LIN {X 0,Y 552.727,Z 232.102,A -85,B 0,C 180,E1 25516.002,E2 25516.002} C_VEL
LIN {X 0,Y 555.255,Z 236.797,A -85,B 0,C 180,E1 25515.534,E2 25515.534} C_VEL
LIN {X 0,Y 562.357,Z 248.705,A -85,B 0,C 180,E1 25514.312,E2 25514.312} C_VEL
LIN {X 0,Y 564.451,Z 252.523,A -85,B 0,C 180,E1 25513.903,E2 25513.903} C_VEL
LIN {X 0,Y 562.986,Z 312.412,A -85,B 0,C 180,E1 25510.976,E2 25510.976} C_VEL
LIN {X 0,Y 564.162,Z 323.504,A -85,B 0,C 180,E1 25510.685,E2 25510.685} C_VEL
LIN {X 0,Y 562.341,Z 534.473,A -85,B 0,C 180,E1 25507.441,E2 25507.441} C_VEL
LIN {X 0,Y 561.246,Z 663.193,A -85,B 0,C 180,E1 25505.485,E2 25505.485} C_VEL
LIN {X 0,Y 560.691,Z 686.814,A -85,B 0,C 180,E1 25504.937,E2 25504.937} C_VEL
LIN {X 0,Y 560.116,Z 709.07,A -85,B 0,C 180,E1 25504.231,E2 25504.231} C_VEL
LIN {X 0,Y 559.344,Z 730.722,A -85,B 0,C 180,E1 25503.343,E2 25503.343} C_VEL
LIN {X 0,Y 558.543,Z 751.818,A -85,B 0,C 180,E1 25502.298,E2 25502.298} C_VEL
LIN {X 0,Y 557.68,Z 772.074,A -85,B 0,C 180,E1 25501.086,E2 25501.086} C_VEL
LIN {X 0,Y 556.797,Z 791.954,A -85,B 0,C 180,E1 25499.709,E2 25499.709} C_VEL
LIN {X 0,Y 555.937,Z 810.881,A -85,B 0,C 180,E1 25498.176,E2 25498.176} C_VEL
LIN {X 0,Y 555.05,Z 830.364,A -85,B 0,C 180,E1 25496.36,E2 25496.36} C_VEL
LIN {X 0,Y 554.323,Z 847.686,A -85,B 0,C 180,E1 25494.509,E2 25494.509} C_VEL
LIN {X 0,Y 553.67,Z 863.855,A -85,B 0,C 180,E1 25492.509,E2 25492.509} C_VEL
LIN {X 0,Y 553.104,Z 879.347,A -85,B 0,C 180,E1 25490.308,E2 25490.308} C_VEL
LIN {X 0,Y 552.685,Z 892.647,A -85,B 0,C 180,E1 25488.128,E2 25488.128} C_VEL
LIN {X 0,Y 552.387,Z 903.847,A -85,B 0,C 180,E1 25485.968,E2 25485.968} C_VEL
LIN {X 0,Y 552.185,Z 913.887,A -85,B 0,C 180,E1 25483.72,E2 25483.72} C_VEL
LIN {X 0,Y 552.045,Z 922.058,A -85,B 0,C 180,E1 25481.491,E2 25481.491} C_VEL
LIN {X 0,Y 551.974,Z 929.049,A -85,B 0,C 180,E1 25479.169,E2 25479.169} C_VEL
LIN {X 0,Y 551.924,Z 934.179,A -85,B 0,C 180,E1 25476.905,E2 25476.905} C_VEL
LIN {X 0,Y 551.901,Z 938.05,A -85,B 0,C 180,E1 25474.571,E2 25474.571} C_VEL
LIN {X 0,Y 551.905,Z 940.19,A -85,B 0,C 180,E1 25472.283,E2 25472.283} C_VEL
LIN {X 0,Y 551.91,Z 940.984,A -85,B 0,C 180,E1 25469.895,E2 25469.895} C_VEL
LIN {X 0,Y 551.905,Z 940.122,A -85,B 0,C 180,E1 25467.611,E2 25467.611} C_VEL
LIN {X 0,Y 551.901,Z 937.911,A -85,B 0,C 180,E1 25465.323,E2 25465.323} C_VEL
LIN {X 0,Y 551.926,Z 934.045,A -85,B 0,C 180,E1 25463.027,E2 25463.027} C_VEL
LIN {X 0,Y 551.977,Z 928.772,A -85,B 0,C 180,E1 25460.722,E2 25460.722} C_VEL
LIN {X 0,Y 552.051,Z 921.694,A -85,B 0,C 180,E1 25458.401,E2 25458.401} C_VEL
LIN {X 0,Y 552.196,Z 912.955,A -85,B 0,C 180,E1 25456.056,E2 25456.056} C_VEL
LIN {X 0,Y 552.397,Z 903.317,A -85,B 0,C 180,E1 25453.922,E2 25453.922} C_VEL
LIN {X 0,Y 552.712,Z 891.365,A -85,B 0,C 180,E1 25451.652,E2 25451.652} C_VEL
LIN {X 0,Y 553.126,Z 878.623,A -85,B 0,C 180,E1 25449.581,E2 25449.581} C_VEL
LIN {X 0,Y 553.701,Z 862.989,A -85,B 0,C 180,E1 25447.378,E2 25447.378} C_VEL
LIN {X 0,Y 554.368,Z 846.587,A -85,B 0,C 180,E1 25445.369,E2 25445.369} C_VEL
LIN {X 0,Y 555.074,Z 829.786,A -85,B 0,C 180,E1 25443.581,E2 25443.581} C_VEL
LIN {X 0,Y 555.964,Z 810.256,A -85,B 0,C 180,E1 25441.771,E2 25441.771} C_VEL
LIN {X 0,Y 556.836,Z 791.177,A -85,B 0,C 180,E1 25440.231,E2 25440.231} C_VEL
LIN {X 0,Y 557.719,Z 771.141,A -85,B 0,C 180,E1 25438.854,E2 25438.854} C_VEL
LIN {X 0,Y 558.61,Z 749.547,A -85,B 0,C 180,E1 25437.582,E2 25437.582} C_VEL
LIN {X 0,Y 559.414,Z 729.067,A -85,B 0,C 180,E1 25436.583,E2 25436.583} C_VEL
LIN {X 0,Y 560.162,Z 706.296,A -85,B 0,C 180,E1 25435.673,E2 25435.673} C_VEL
LIN {X 0,Y 560.75,Z 685.166,A -85,B 0,C 180,E1 25435.018,E2 25435.018} C_VEL
LIN {X 0,Y 561.258,Z 661.984,A -85,B 0,C 180,E1 25434.493,E2 25434.493} C_VEL
LIN {X 0,Y 563.081,Z 445.342,A -85,B 0,C 180,E1 25431.201,E2 25431.201} C_VEL
LIN {X 0,Y 564.019,Z 320.67,A -85,B 0,C 180,E1 25429.256,E2 25429.256} C_VEL
LIN {X 0,Y 562.94,Z 311.331,A -85,B 0,C 180,E1 25428.982,E2 25428.982} C_VEL
LIN {X 0,Y 564.451,Z 252.523,A -85,B 0,C 180,E1 25426.097,E2 25426.097} C_VEL
LIN {X 0,Y 557.462,Z 240.492,A -85,B 0,C 180,E1 25424.82,E2 25424.82} C_VEL
LIN {X 0,Y 553.879,Z 234.143,A -85,B 0,C 180,E1 25424.171,E2 25424.171} C_VEL
LIN {X 0,Y 552.316,Z 230.647,A -85,B 0,C 180,E1 25423.789,E2 25423.789} C_VEL
LIN {X 0,Y 552.267,Z 230.221,A -85,B 0,C 180,E1 25423.296,E2 25423.296} C_VEL
LIN {X 0,Y 552.269,Z 230.249,A -85,B 0,C 180,E1 25419.994,E2 25419.994} C_VEL
LIN {X 0,Y 552.295,Z 230.247,A -85,B 0,C 180,E1 25416.945,E2 25416.945} C_VEL
LIN {X 0,Y 552.268,Z 230.252,A -85,B 0,C 180,E1 25413.642,E2 25413.642} C_VEL
LIN {X 0,Y 552.343,Z 230.249,A -85,B 0,C 180,E1 25410.455,E2 25410.455} C_VEL
LIN {X 0,Y 552.273,Z 230.251,A -85,B 0,C 180,E1 25407.26,E2 25407.26} C_VEL
LIN {X 0,Y 552.324,Z 230.248,A -85,B 0,C 180,E1 25404.036,E2 25404.036} C_VEL
LIN {X 0,Y 552.287,Z 230.248,A -85,B 0,C 180,E1 25400.895,E2 25400.895} C_VEL
LIN {X 0,Y 552.288,Z 230.247,A -85,B 0,C 180,E1 25397.43,E2 25397.43} C_VEL
LIN {X 0,Y 552.339,Z 230.243,A -85,B 0,C 180,E1 25394.252,E2 25394.252} C_VEL
LIN {X 0,Y 552.286,Z 230.246,A -85,B 0,C 180,E1 25390.958,E2 25390.958} C_VEL
LIN {X 0,Y 552.34,Z 230.243,A -85,B 0,C 180,E1 25387.699,E2 25387.699} C_VEL
LIN {X 0,Y 552.304,Z 230.245,A -85,B 0,C 180,E1 25384.465,E2 25384.465} C_VEL
LIN {X 0,Y 552.3,Z 230.238,A -85,B 0,C 180,E1 25381.038,E2 25381.038} C_VEL
LIN {X 0,Y 552.342,Z 230.244,A -85,B 0,C 180,E1 25377.774,E2 25377.774} C_VEL
LIN {X 0,Y 552.301,Z 230.245,A -85,B 0,C 180,E1 25374.495,E2 25374.495} C_VEL
LIN {X 0,Y 552.332,Z 230.236,A -85,B 0,C 180,E1 25371.149,E2 25371.149} C_VEL
LIN {X 0,Y 552.338,Z 230.247,A -85,B 0,C 180,E1 25367.773,E2 25367.773} C_VEL
LIN {X 0,Y 552.307,Z 230.243,A -85,B 0,C 180,E1 25364.459,E2 25364.459} C_VEL
LIN {X 0,Y 552.34,Z 230.235,A -85,B 0,C 180,E1 25361.203,E2 25361.203} C_VEL
LIN {X 0,Y 552.324,Z 230.248,A -85,B 0,C 180,E1 25357.881,E2 25357.881} C_VEL
LIN {X 0,Y 552.322,Z 230.24,A -85,B 0,C 180,E1 25354.479,E2 25354.479} C_VEL
LIN {X 0,Y 552.34,Z 230.241,A -85,B 0,C 180,E1 25352.776,E2 25352.776} C_VEL
LIN {X 0,Y 551.359,Z 230.367,A -85,B 0,C 180,E1 25351.977,E2 25351.977} C_VEL
LIN {X 0,Y 544.843,Z 231.184,A -85,B 0,C 180,E1 25349.675,E2 25349.675} C_VEL
LIN {X 0,Y 544.396,Z 231.235,A -85,B 0,C 180,E1 25349.149,E2 25349.149} C_VEL
LIN {X 0,Y 544.387,Z 231.233,A -85,B 0,C 180,E1 25345.742,E2 25345.742} C_VEL
LIN {X 0,Y 544.395,Z 231.23,A -85,B 0,C 180,E1 25342.295,E2 25342.295} C_VEL
LIN {X 0,Y 544.391,Z 231.235,A -85,B 0,C 180,E1 25338.89,E2 25338.89} C_VEL
LIN {X 0,Y 544.389,Z 231.229,A -85,B 0,C 180,E1 25335.593,E2 25335.593} C_VEL
LIN {X 0,Y 544.399,Z 231.227,A -85,B 0,C 180,E1 25332.238,E2 25332.238} C_VEL
LIN {X 0,Y 544.387,Z 231.234,A -85,B 0,C 180,E1 25328.779,E2 25328.779} C_VEL
LIN {X 0,Y 544.393,Z 231.234,A -85,B 0,C 180,E1 25325.478,E2 25325.478} C_VEL
LIN {X 0,Y 544.39,Z 231.232,A -85,B 0,C 180,E1 25322.147,E2 25322.147} C_VEL
LIN {X 0,Y 544.385,Z 231.238,A -85,B 0,C 180,E1 25318.645,E2 25318.645} C_VEL
LIN {X 0,Y 544.397,Z 231.232,A -85,B 0,C 180,E1 25315.338,E2 25315.338} C_VEL
LIN {X 0,Y 544.375,Z 231.209,A -85,B 0,C 180,E1 25312.006,E2 25312.006} C_VEL
LIN {X 0,Y 544.383,Z 231.233,A -85,B 0,C 180,E1 25308.528,E2 25308.528} C_VEL
LIN {X 0,Y 544.401,Z 231.228,A -85,B 0,C 180,E1 25305.118,E2 25305.118} C_VEL
LIN {X 0,Y 544.37,Z 231.209,A -85,B 0,C 180,E1 25301.774,E2 25301.774} C_VEL
LIN {X 0,Y 544.447,Z 231.538,A -85,B 0,C 180,E1 25301.255,E2 25301.255} C_VEL
LIN {X 0,Y 545.979,Z 235.096,A -85,B 0,C 180,E1 25300.825,E2 25300.825} C_VEL
LIN {X 0,Y 553.743,Z 252.148,A -85,B 0,C 180,E1 25299.008,E2 25299.008} C_VEL
LIN {X 0,Y 551.806,Z 305.653,A -85,B 0,C 180,E1 25295.668,E2 25295.668} C_VEL
LIN {X 0,Y 550.042,Z 360.38,A -85,B 0,C 180,E1 25292.345,E2 25292.345} C_VEL
LIN {X 0,Y 548.57,Z 416.762,A -85,B 0,C 180,E1 25289.006,E2 25289.006} C_VEL
LIN {X 0,Y 549.487,Z 426.879,A -85,B 0,C 180,E1 25288.789,E2 25288.789} C_VEL
LIN {X 0,Y 547.988,Z 628.997,A -85,B 0,C 180,E1 25285.906,E2 25285.906} C_VEL
LIN {X 0,Y 547.682,Z 647.765,A -85,B 0,C 180,E1 25285.445,E2 25285.445} C_VEL
LIN {X 0,Y 547.303,Z 665.668,A -85,B 0,C 180,E1 25284.813,E2 25284.813} C_VEL
LIN {X 0,Y 546.844,Z 682.777,A -85,B 0,C 180,E1 25284.019,E2 25284.019} C_VEL
LIN {X 0,Y 546.339,Z 699.932,A -85,B 0,C 180,E1 25283.011,E2 25283.011} C_VEL
LIN {X 0,Y 545.837,Z 716.086,A -85,B 0,C 180,E1 25281.84,E2 25281.84} C_VEL
LIN {X 0,Y 545.354,Z 731.27,A -85,B 0,C 180,E1 25280.504,E2 25280.504} C_VEL
LIN {X 0,Y 544.923,Z 745.434,A -85,B 0,C 180,E1 25279,E2 25279} C_VEL
LIN {X 0,Y 544.573,Z 758.1,A -85,B 0,C 180,E1 25277.381,E2 25277.381} C_VEL
LIN {X 0,Y 544.3,Z 769.323,A -85,B 0,C 180,E1 25275.643,E2 25275.643} C_VEL
LIN {X 0,Y 544.122,Z 778.555,A -85,B 0,C 180,E1 25273.892,E2 25273.892} C_VEL
LIN {X 0,Y 544,Z 786.466,A -85,B 0,C 180,E1 25272.016,E2 25272.016} C_VEL
LIN {X 0,Y 543.946,Z 792.587,A -85,B 0,C 180,E1 25270.121,E2 25270.121} C_VEL
LIN {X 0,Y 543.915,Z 797.083,A -85,B 0,C 180,E1 25268.172,E2 25268.172} C_VEL
LIN {X 0,Y 543.916,Z 799.805,A -85,B 0,C 180,E1 25266.262,E2 25266.262} C_VEL
LIN {X 0,Y 543.913,Z 800.941,A -85,B 0,C 180,E1 25264.255,E2 25264.255} C_VEL
LIN {X 0,Y 543.911,Z 800.358,A -85,B 0,C 180,E1 25262.286,E2 25262.286} C_VEL
LIN {X 0,Y 543.914,Z 798.153,A -85,B 0,C 180,E1 25260.365,E2 25260.365} C_VEL
LIN {X 0,Y 543.933,Z 794.203,A -85,B 0,C 180,E1 25258.408,E2 25258.408} C_VEL
LIN {X 0,Y 543.974,Z 788.738,A -85,B 0,C 180,E1 25256.537,E2 25256.537} C_VEL
LIN {X 0,Y 544.075,Z 781.346,A -85,B 0,C 180,E1 25254.63,E2 25254.63} C_VEL
LIN {X 0,Y 544.237,Z 772.416,A -85,B 0,C 180,E1 25252.814,E2 25252.814} C_VEL
LIN {X 0,Y 544.471,Z 762.018,A -85,B 0,C 180,E1 25251.096,E2 25251.096} C_VEL
LIN {X 0,Y 544.794,Z 749.92,A -85,B 0,C 180,E1 25249.446,E2 25249.446} C_VEL
LIN {X 0,Y 545.205,Z 736.375,A -85,B 0,C 180,E1 25247.912,E2 25247.912} C_VEL
LIN {X 0,Y 545.673,Z 721.557,A -85,B 0,C 180,E1 25246.518,E2 25246.518} C_VEL
LIN {X 0,Y 546.19,Z 705.24,A -85,B 0,C 180,E1 25245.256,E2 25245.256} C_VEL
LIN {X 0,Y 546.683,Z 688.447,A -85,B 0,C 180,E1 25244.199,E2 25244.199} C_VEL
LIN {X 0,Y 547.148,Z 671.418,A -85,B 0,C 180,E1 25243.341,E2 25243.341} C_VEL
LIN {X 0,Y 547.569,Z 653.244,A -85,B 0,C 180,E1 25242.638,E2 25242.638} C_VEL
LIN {X 0,Y 547.905,Z 634.586,A -85,B 0,C 180,E1 25242.122,E2 25242.122} C_VEL
LIN {X 0,Y 548.12,Z 613.896,A -85,B 0,C 180,E1 25241.767,E2 25241.767} C_VEL
LIN {X 0,Y 549.615,Z 423.975,A -85,B 0,C 180,E1 25239.038,E2 25239.038} C_VEL
LIN {X 0,Y 548.63,Z 415.642,A -85,B 0,C 180,E1 25238.823,E2 25238.823} C_VEL
LIN {X 0,Y 550.36,Z 360.162,A -85,B 0,C 180,E1 25235.488,E2 25235.488} C_VEL
LIN {X 0,Y 552.396,Z 305.248,A -85,B 0,C 180,E1 25232.106,E2 25232.106} C_VEL
LIN {X 0,Y 554.6,Z 253.28,A -85,B 0,C 180,E1 25228.819,E2 25228.819} C_VEL
LIN {X 0,Y 546.033,Z 235.235,A -85,B 0,C 180,E1 25226.772,E2 25226.772} C_VEL
LIN {X 0,Y 544.394,Z 231.707,A -85,B 0,C 180,E1 25226.33,E2 25226.33} C_VEL
LIN {X 0,Y 544.322,Z 231.245,A -85,B 0,C 180,E1 25226.04,E2 25226.04} C_VEL
LIN {X 0,Y 544.349,Z 231.241,A -85,B 0,C 180,E1 25222.688,E2 25222.688} C_VEL
LIN {X 0,Y 544.333,Z 231.242,A -85,B 0,C 180,E1 25219.642,E2 25219.642} C_VEL
LIN {X 0,Y 544.325,Z 231.242,A -85,B 0,C 180,E1 25216.212,E2 25216.212} C_VEL
LIN {X 0,Y 544.358,Z 231.241,A -85,B 0,C 180,E1 25213.165,E2 25213.165} C_VEL
LIN {X 0,Y 544.32,Z 231.24,A -85,B 0,C 180,E1 25209.942,E2 25209.942} C_VEL
LIN {X 0,Y 544.392,Z 231.237,A -85,B 0,C 180,E1 25206.75,E2 25206.75} C_VEL
LIN {X 0,Y 544.317,Z 231.241,A -85,B 0,C 180,E1 25203.475,E2 25203.475} C_VEL
LIN {X 0,Y 544.36,Z 231.237,A -85,B 0,C 180,E1 25200.21,E2 25200.21} C_VEL
LIN {X 0,Y 544.321,Z 231.24,A -85,B 0,C 180,E1 25197.157,E2 25197.157} C_VEL
LIN {X 0,Y 544.334,Z 231.239,A -85,B 0,C 180,E1 25193.778,E2 25193.778} C_VEL
LIN {X 0,Y 544.331,Z 231.239,A -85,B 0,C 180,E1 25190.804,E2 25190.804} C_VEL
LIN {X 0,Y 544.319,Z 231.24,A -85,B 0,C 180,E1 25187.373,E2 25187.373} C_VEL
LIN {X 0,Y 544.375,Z 231.236,A -85,B 0,C 180,E1 25184.226,E2 25184.226} C_VEL
LIN {X 0,Y 544.316,Z 231.241,A -85,B 0,C 180,E1 25181.026,E2 25181.026} C_VEL
LIN {X 0,Y 544.383,Z 231.238,A -85,B 0,C 180,E1 25177.768,E2 25177.768} C_VEL
LIN {X 0,Y 544.319,Z 231.24,A -85,B 0,C 180,E1 25174.652,E2 25174.652} C_VEL
LIN {X 0,Y 544.353,Z 231.242,A -85,B 0,C 180,E1 25171.354,E2 25171.354} C_VEL
LIN {X 0,Y 544.326,Z 231.242,A -85,B 0,C 180,E1 25168.308,E2 25168.308} C_VEL
LIN {X 0,Y 544.326,Z 231.243,A -85,B 0,C 180,E1 25164.823,E2 25164.823} C_VEL
LIN {X 0,Y 544.377,Z 231.239,A -85,B 0,C 180,E1 25161.625,E2 25161.625} C_VEL
LIN {X 0,Y 544.318,Z 231.243,A -85,B 0,C 180,E1 25158.382,E2 25158.382} C_VEL
LIN {X 0,Y 544.367,Z 231.373,A -85,B 0,C 180,E1 25156.901,E2 25156.901} C_VEL
LIN {X 0,Y 544.631,Z 232.618,A -85,B 0,C 180,E1 25156.71,E2 25156.71} C_VEL
LIN {X 0,Y 556.335,Z 253.338,A -85,B 0,C 180,E1 25154.627,E2 25154.627} C_VEL
LIN {X 0,Y 558.328,Z 256.699,A -85,B 0,C 180,E1 25154.287,E2 25154.287} C_VEL
LIN {X 0,Y 556.801,Z 312.976,A -85,B 0,C 180,E1 25151.517,E2 25151.517} C_VEL
LIN {X 0,Y 558.08,Z 324.936,A -85,B 0,C 180,E1 25151.2,E2 25151.2} C_VEL
LIN {X 0,Y 555.975,Z 535.872,A -85,B 0,C 180,E1 25147.923,E2 25147.923} C_VEL
LIN {X 0,Y 554.725,Z 663.15,A -85,B 0,C 180,E1 25145.968,E2 25145.968} C_VEL
LIN {X 0,Y 554.109,Z 686.682,A -85,B 0,C 180,E1 25145.418,E2 25145.418} C_VEL
LIN {X 0,Y 553.432,Z 708.705,A -85,B 0,C 180,E1 25144.716,E2 25144.716} C_VEL
LIN {X 0,Y 552.599,Z 729.782,A -85,B 0,C 180,E1 25143.85,E2 25143.85} C_VEL
LIN {X 0,Y 551.715,Z 749.594,A -85,B 0,C 180,E1 25142.871,E2 25142.871} C_VEL
LIN {X 0,Y 550.684,Z 771.086,A -85,B 0,C 180,E1 25141.593,E2 25141.593} C_VEL
LIN {X 0,Y 549.669,Z 791.21,A -85,B 0,C 180,E1 25140.194,E2 25140.194} C_VEL
LIN {X 0,Y 548.625,Z 810.875,A -85,B 0,C 180,E1 25138.586,E2 25138.586} C_VEL
LIN {X 0,Y 547.59,Z 830.219,A -85,B 0,C 180,E1 25136.763,E2 25136.763} C_VEL
LIN {X 0,Y 546.756,Z 847.686,A -85,B 0,C 180,E1 25134.871,E2 25134.871} C_VEL
LIN {X 0,Y 545.977,Z 863.853,A -85,B 0,C 180,E1 25132.844,E2 25132.844} C_VEL
LIN {X 0,Y 545.309,Z 879.349,A -85,B 0,C 180,E1 25130.611,E2 25130.611} C_VEL
LIN {X 0,Y 544.822,Z 892.645,A -85,B 0,C 180,E1 25128.399,E2 25128.399} C_VEL
LIN {X 0,Y 544.469,Z 904.015,A -85,B 0,C 180,E1 25126.172,E2 25126.172} C_VEL
LIN {X 0,Y 544.223,Z 914.298,A -85,B 0,C 180,E1 25123.817,E2 25123.817} C_VEL
LIN {X 0,Y 544.066,Z 922.415,A -85,B 0,C 180,E1 25121.554,E2 25121.554} C_VEL
LIN {X 0,Y 543.974,Z 929.554,A -85,B 0,C 180,E1 25119.094,E2 25119.094} C_VEL
LIN {X 0,Y 543.928,Z 934.274,A -85,B 0,C 180,E1 25116.958,E2 25116.958} C_VEL
LIN {X 0,Y 543.901,Z 938.05,A -85,B 0,C 180,E1 25114.638,E2 25114.638} C_VEL
LIN {X 0,Y 543.905,Z 940.19,A -85,B 0,C 180,E1 25112.317,E2 25112.317} C_VEL
LIN {X 0,Y 543.91,Z 940.984,A -85,B 0,C 180,E1 25109.894,E2 25109.894} C_VEL
LIN {X 0,Y 543.907,Z 940.122,A -85,B 0,C 180,E1 25107.576,E2 25107.576} C_VEL
LIN {X 0,Y 543.903,Z 937.912,A -85,B 0,C 180,E1 25105.254,E2 25105.254} C_VEL
LIN {X 0,Y 543.932,Z 934.046,A -85,B 0,C 180,E1 25102.924,E2 25102.924} C_VEL
LIN {X 0,Y 543.983,Z 928.772,A -85,B 0,C 180,E1 25100.584,E2 25100.584} C_VEL
LIN {X 0,Y 544.072,Z 921.694,A -85,B 0,C 180,E1 25098.229,E2 25098.229} C_VEL
LIN {X 0,Y 544.247,Z 912.99,A -85,B 0,C 180,E1 25095.856,E2 25095.856} C_VEL
LIN {X 0,Y 544.487,Z 903.319,A -85,B 0,C 180,E1 25093.682,E2 25093.682} C_VEL
LIN {X 0,Y 544.862,Z 891.364,A -85,B 0,C 180,E1 25091.378,E2 25091.378} C_VEL
LIN {X 0,Y 545.335,Z 878.625,A -85,B 0,C 180,E1 25089.275,E2 25089.275} C_VEL
LIN {X 0,Y 545.999,Z 863.35,A -85,B 0,C 180,E1 25087.09,E2 25087.09} C_VEL
LIN {X 0,Y 546.77,Z 847.396,A -85,B 0,C 180,E1 25085.096,E2 25085.096} C_VEL
LIN {X 0,Y 547.59,Z 830.217,A -85,B 0,C 180,E1 25083.237,E2 25083.237} C_VEL
LIN {X 0,Y 548.624,Z 810.87,A -85,B 0,C 180,E1 25081.414,E2 25081.414} C_VEL
LIN {X 0,Y 549.67,Z 791.175,A -85,B 0,C 180,E1 25079.803,E2 25079.803} C_VEL
LIN {X 0,Y 550.704,Z 770.626,A -85,B 0,C 180,E1 25078.377,E2 25078.377} C_VEL
LIN {X 0,Y 551.717,Z 749.551,A -85,B 0,C 180,E1 25077.126,E2 25077.126} C_VEL
LIN {X 0,Y 552.617,Z 729.382,A -85,B 0,C 180,E1 25076.132,E2 25076.132} C_VEL
LIN {X 0,Y 553.473,Z 706.678,A -85,B 0,C 180,E1 25075.213,E2 25075.213} C_VEL
LIN {X 0,Y 554.157,Z 685.425,A -85,B 0,C 180,E1 25074.547,E2 25074.547} C_VEL
LIN {X 0,Y 554.735,Z 662.276,A -85,B 0,C 180,E1 25074.017,E2 25074.017} C_VEL
LIN {X 0,Y 556.825,Z 447.482,A -85,B 0,C 180,E1 25070.717,E2 25070.717} C_VEL
LIN {X 0,Y 557.939,Z 322.075,A -85,B 0,C 180,E1 25068.739,E2 25068.739} C_VEL
LIN {X 0,Y 556.709,Z 311.331,A -85,B 0,C 180,E1 25068.422,E2 25068.422} C_VEL
LIN {X 0,Y 558.314,Z 256.678,A -85,B 0,C 180,E1 25065.711,E2 25065.711} C_VEL
LIN {X 0,Y 546.636,Z 236.072,A -85,B 0,C 180,E1 25063.597,E2 25063.597} C_VEL
LIN {X 0,Y 544.539,Z 232.255,A -85,B 0,C 180,E1 25063.178,E2 25063.178} C_VEL
LIN {X 0,Y 544.367,Z 231.262,A -85,B 0,C 180,E1 25062.955,E2 25062.955} C_VEL
LIN {X 0,Y 544.321,Z 231.237,A -85,B 0,C 180,E1 25059.735,E2 25059.735} C_VEL
LIN {X 0,Y 544.391,Z 231.236,A -85,B 0,C 180,E1 25056.518,E2 25056.518} C_VEL
LIN {X 0,Y 544.329,Z 231.242,A -85,B 0,C 180,E1 25053.303,E2 25053.303} C_VEL
LIN {X 0,Y 544.357,Z 231.237,A -85,B 0,C 180,E1 25049.974,E2 25049.974} C_VEL
LIN {X 0,Y 544.346,Z 231.241,A -85,B 0,C 180,E1 25046.981,E2 25046.981} C_VEL
LIN {X 0,Y 544.344,Z 231.238,A -85,B 0,C 180,E1 25043.569,E2 25043.569} C_VEL
LIN {X 0,Y 544.391,Z 231.239,A -85,B 0,C 180,E1 25040.424,E2 25040.424} C_VEL
LIN {X 0,Y 544.343,Z 231.237,A -85,B 0,C 180,E1 25037.091,E2 25037.091} C_VEL
LIN {X 0,Y 544.393,Z 231.234,A -85,B 0,C 180,E1 25033.814,E2 25033.814} C_VEL
LIN {X 0,Y 544.361,Z 231.236,A -85,B 0,C 180,E1 25030.584,E2 25030.584} C_VEL
LIN {X 0,Y 544.356,Z 231.234,A -85,B 0,C 180,E1 25027.175,E2 25027.175} C_VEL
LIN {X 0,Y 544.406,Z 231.237,A -85,B 0,C 180,E1 25023.897,E2 25023.897} C_VEL
LIN {X 0,Y 544.357,Z 231.228,A -85,B 0,C 180,E1 25020.632,E2 25020.632} C_VEL
LIN {X 0,Y 544.386,Z 231.228,A -85,B 0,C 180,E1 25017.263,E2 25017.263} C_VEL
LIN {X 0,Y 544.401,Z 231.238,A -85,B 0,C 180,E1 25013.885,E2 25013.885} C_VEL
LIN {X 0,Y 544.365,Z 231.227,A -85,B 0,C 180,E1 25010.592,E2 25010.592} C_VEL
LIN {X 0,Y 544.403,Z 231.227,A -85,B 0,C 180,E1 25007.226,E2 25007.226} C_VEL
LIN {X 0,Y 544.396,Z 231.237,A -85,B 0,C 180,E1 25003.79,E2 25003.79} C_VEL
LIN {X 0,Y 544.372,Z 231.225,A -85,B 0,C 180,E1 25000.432,E2 25000.432} C_VEL
LIN {X 0,Y 544.4,Z 231.229,A -85,B 0,C 180,E1 24997.086,E2 24997.086} C_VEL
LIN {X 0,Y 544.395,Z 231.235,A -85,B 0,C 180,E1 24993.674,E2 24993.674} C_VEL
LIN {X 0,Y 544.381,Z 231.224,A -85,B 0,C 180,E1 24990.271,E2 24990.271} C_VEL
LIN {X 0,Y 544.396,Z 231.235,A -85,B 0,C 180,E1 24989.149,E2 24989.149} C_VEL
LIN {X 0,Y 543.394,Z 231.356,A -85,B 0,C 180,E1 24988.338,E2 24988.338} C_VEL
LIN {X 0,Y 536.981,Z 232.155,A -85,B 0,C 180,E1 24986.061,E2 24986.061} C_VEL
LIN {X 0,Y 536.459,Z 232.218,A -85,B 0,C 180,E1 24985.468,E2 24985.468} C_VEL
LIN {X 0,Y 536.447,Z 232.222,A -85,B 0,C 180,E1 24982.038,E2 24982.038} C_VEL
LIN {X 0,Y 536.453,Z 232.222,A -85,B 0,C 180,E1 24978.689,E2 24978.689} C_VEL
LIN {X 0,Y 536.46,Z 232.219,A -85,B 0,C 180,E1 24975.21,E2 24975.21} C_VEL
LIN {X 0,Y 536.451,Z 232.218,A -85,B 0,C 180,E1 24971.796,E2 24971.796} C_VEL
LIN {X 0,Y 536.447,Z 232.22,A -85,B 0,C 180,E1 24968.482,E2 24968.482} C_VEL
LIN {X 0,Y 536.462,Z 232.226,A -85,B 0,C 180,E1 24965.034,E2 24965.034} C_VEL
LIN {X 0,Y 536.458,Z 232.222,A -85,B 0,C 180,E1 24961.584,E2 24961.584} C_VEL
LIN {X 0,Y 536.446,Z 232.223,A -85,B 0,C 180,E1 24958.165,E2 24958.165} C_VEL
LIN {X 0,Y 536.451,Z 232.226,A -85,B 0,C 180,E1 24954.678,E2 24954.678} C_VEL
LIN {X 0,Y 536.457,Z 232.194,A -85,B 0,C 180,E1 24951.268,E2 24951.268} C_VEL
LIN {X 0,Y 536.438,Z 232.217,A -85,B 0,C 180,E1 24947.912,E2 24947.912} C_VEL
LIN {X 0,Y 536.444,Z 232.23,A -85,B 0,C 180,E1 24944.464,E2 24944.464} C_VEL
LIN {X 0,Y 536.464,Z 232.463,A -85,B 0,C 180,E1 24941.941,E2 24941.941} C_VEL
LIN {X 0,Y 537.463,Z 235.23,A -85,B 0,C 180,E1 24941.591,E2 24941.591} C_VEL
LIN {X 0,Y 540.592,Z 241.643,A -85,B 0,C 180,E1 24940.857,E2 24940.857} C_VEL
LIN {X 0,Y 547.048,Z 255.602,A -85,B 0,C 180,E1 24939.336,E2 24939.336} C_VEL
LIN {X 0,Y 544.995,Z 307.604,A -85,B 0,C 180,E1 24936.056,E2 24936.056} C_VEL
LIN {X 0,Y 543.029,Z 362.364,A -85,B 0,C 180,E1 24932.692,E2 24932.692} C_VEL
LIN {X 0,Y 541.472,Z 416.047,A -85,B 0,C 180,E1 24929.479,E2 24929.479} C_VEL
LIN {X 0,Y 542.652,Z 427.737,A -85,B 0,C 180,E1 24929.218,E2 24929.218} C_VEL
LIN {X 0,Y 540.797,Z 628.637,A -85,B 0,C 180,E1 24926.284,E2 24926.284} C_VEL
LIN {X 0,Y 540.393,Z 647.439,A -85,B 0,C 180,E1 24925.81,E2 24925.81} C_VEL
LIN {X 0,Y 539.894,Z 665.243,A -85,B 0,C 180,E1 24925.162,E2 24925.162} C_VEL
LIN {X 0,Y 539.28,Z 682.941,A -85,B 0,C 180,E1 24924.309,E2 24924.309} C_VEL
LIN {X 0,Y 538.667,Z 700.782,A -85,B 0,C 180,E1 24923.234,E2 24923.234} C_VEL
LIN {X 0,Y 538.098,Z 716.848,A -85,B 0,C 180,E1 24922.042,E2 24922.042} C_VEL
LIN {X 0,Y 537.534,Z 732.437,A -85,B 0,C 180,E1 24920.634,E2 24920.634} C_VEL
LIN {X 0,Y 537.063,Z 745.957,A -85,B 0,C 180,E1 24919.163,E2 24919.163} C_VEL
LIN {X 0,Y 536.665,Z 758.537,A -85,B 0,C 180,E1 24917.52,E2 24917.52} C_VEL
LIN {X 0,Y 536.36,Z 769.563,A -85,B 0,C 180,E1 24915.777,E2 24915.777} C_VEL
LIN {X 0,Y 536.152,Z 778.846,A -85,B 0,C 180,E1 24913.98,E2 24913.98} C_VEL
LIN {X 0,Y 536.014,Z 786.694,A -85,B 0,C 180,E1 24912.076,E2 24912.076} C_VEL
LIN {X 0,Y 535.95,Z 792.758,A -85,B 0,C 180,E1 24910.153,E2 24910.153} C_VEL
LIN {X 0,Y 535.916,Z 797.137,A -85,B 0,C 180,E1 24908.207,E2 24908.207} C_VEL
LIN {X 0,Y 535.916,Z 799.869,A -85,B 0,C 180,E1 24906.236,E2 24906.236} C_VEL
LIN {X 0,Y 535.913,Z 800.946,A -85,B 0,C 180,E1 24904.235,E2 24904.235} C_VEL
LIN {X 0,Y 535.91,Z 800.318,A -85,B 0,C 180,E1 24902.199,E2 24902.199} C_VEL
LIN {X 0,Y 535.918,Z 798.057,A -85,B 0,C 180,E1 24900.248,E2 24900.248} C_VEL
LIN {X 0,Y 535.937,Z 794.045,A -85,B 0,C 180,E1 24898.259,E2 24898.259} C_VEL
LIN {X 0,Y 535.996,Z 788.327,A -85,B 0,C 180,E1 24896.301,E2 24896.301} C_VEL
LIN {X 0,Y 536.107,Z 780.982,A -85,B 0,C 180,E1 24894.404,E2 24894.404} C_VEL
LIN {X 0,Y 536.301,Z 772.023,A -85,B 0,C 180,E1 24892.573,E2 24892.573} C_VEL
LIN {X 0,Y 536.578,Z 761.478,A -85,B 0,C 180,E1 24890.819,E2 24890.819} C_VEL
LIN {X 0,Y 536.948,Z 749.603,A -85,B 0,C 180,E1 24889.188,E2 24889.188} C_VEL
LIN {X 0,Y 537.432,Z 735.793,A -85,B 0,C 180,E1 24887.611,E2 24887.611} C_VEL
LIN {X 0,Y 537.968,Z 720.886,A -85,B 0,C 180,E1 24886.202,E2 24886.202} C_VEL
LIN {X 0,Y 538.548,Z 704.63,A -85,B 0,C 180,E1 24884.938,E2 24884.938} C_VEL
LIN {X 0,Y 539.121,Z 687.84,A -85,B 0,C 180,E1 24883.874,E2 24883.874} C_VEL
LIN {X 0,Y 539.767,Z 669.679,A -85,B 0,C 180,E1 24882.935,E2 24882.935} C_VEL
LIN {X 0,Y 540.326,Z 651.606,A -85,B 0,C 180,E1 24882.222,E2 24882.222} C_VEL
LIN {X 0,Y 540.779,Z 632.692,A -85,B 0,C 180,E1 24881.696,E2 24881.696} C_VEL
LIN {X 0,Y 541.176,Z 604.747,A -85,B 0,C 180,E1 24881.23,E2 24881.23} C_VEL
LIN {X 0,Y 542.895,Z 424.489,A -85,B 0,C 180,E1 24878.57,E2 24878.57} C_VEL
LIN {X 0,Y 541.632,Z 414.438,A -85,B 0,C 180,E1 24878.3,E2 24878.3} C_VEL
LIN {X 0,Y 543.618,Z 358.391,A -85,B 0,C 180,E1 24874.887,E2 24874.887} C_VEL
LIN {X 0,Y 545.855,Z 303.633,A -85,B 0,C 180,E1 24871.469,E2 24871.469} C_VEL
LIN {X 0,Y 548.025,Z 256.919,A -85,B 0,C 180,E1 24868.481,E2 24868.481} C_VEL
LIN {X 0,Y 539.854,Z 239.957,A -85,B 0,C 180,E1 24866.509,E2 24866.509} C_VEL
LIN {X 0,Y 537.872,Z 235.977,A -85,B 0,C 180,E1 24866.021,E2 24866.021} C_VEL
LIN {X 0,Y 536.455,Z 232.517,A -85,B 0,C 180,E1 24865.57,E2 24865.57} C_VEL
LIN {X 0,Y 536.38,Z 232.219,A -85,B 0,C 180,E1 24864.21,E2 24864.21} C_VEL
LIN {X 0,Y 536.448,Z 232.213,A -85,B 0,C 180,E1 24860.968,E2 24860.968} C_VEL
LIN {X 0,Y 536.387,Z 232.232,A -85,B 0,C 180,E1 24857.688,E2 24857.688} C_VEL
LIN {X 0,Y 536.391,Z 232.231,A -85,B 0,C 180,E1 24854.24,E2 24854.24} C_VEL
LIN {X 0,Y 536.425,Z 232.23,A -85,B 0,C 180,E1 24851.068,E2 24851.068} C_VEL
LIN {X 0,Y 536.379,Z 232.226,A -85,B 0,C 180,E1 24847.821,E2 24847.821} C_VEL
LIN {X 0,Y 536.449,Z 232.225,A -85,B 0,C 180,E1 24844.596,E2 24844.596} C_VEL
LIN {X 0,Y 536.38,Z 232.23,A -85,B 0,C 180,E1 24841.388,E2 24841.388} C_VEL
LIN {X 0,Y 536.412,Z 232.229,A -85,B 0,C 180,E1 24838.077,E2 24838.077} C_VEL
LIN {X 0,Y 536.388,Z 232.231,A -85,B 0,C 180,E1 24834.973,E2 24834.973} C_VEL
LIN {X 0,Y 536.382,Z 232.228,A -85,B 0,C 180,E1 24831.531,E2 24831.531} C_VEL
LIN {X 0,Y 536.441,Z 232.226,A -85,B 0,C 180,E1 24828.278,E2 24828.278} C_VEL
LIN {X 0,Y 536.375,Z 232.226,A -85,B 0,C 180,E1 24825.093,E2 24825.093} C_VEL
LIN {X 0,Y 536.438,Z 232.226,A -85,B 0,C 180,E1 24821.864,E2 24821.864} C_VEL
LIN {X 0,Y 536.381,Z 232.228,A -85,B 0,C 180,E1 24818.685,E2 24818.685} C_VEL
LIN {X 0,Y 536.399,Z 232.23,A -85,B 0,C 180,E1 24815.32,E2 24815.32} C_VEL
LIN {X 0,Y 536.401,Z 232.231,A -85,B 0,C 180,E1 24812.225,E2 24812.225} C_VEL
LIN {X 0,Y 536.385,Z 232.231,A -85,B 0,C 180,E1 24808.912,E2 24808.912} C_VEL
LIN {X 0,Y 536.437,Z 232.228,A -85,B 0,C 180,E1 24805.744,E2 24805.744} C_VEL
LIN {X 0,Y 536.38,Z 232.234,A -85,B 0,C 180,E1 24802.442,E2 24802.442} C_VEL
LIN {X 0,Y 536.427,Z 232.215,A -85,B 0,C 180,E1 24799.138,E2 24799.138} C_VEL
LIN {X 0,Y 536.466,Z 232.475,A -85,B 0,C 180,E1 24797.564,E2 24797.564} C_VEL
LIN {X 0,Y 537.007,Z 234.315,A -85,B 0,C 180,E1 24797.333,E2 24797.333} C_VEL
LIN {X 0,Y 538.981,Z 237.919,A -85,B 0,C 180,E1 24796.947,E2 24796.947} C_VEL
LIN {X 0,Y 550.927,Z 259.003,A -85,B 0,C 180,E1 24794.797,E2 24794.797} C_VEL
LIN {X 0,Y 551.867,Z 260.567,A -85,B 0,C 180,E1 24794.641,E2 24794.641} C_VEL
LIN {X 0,Y 551.041,Z 295.958,A -85,B 0,C 180,E1 24792.911,E2 24792.911} C_VEL
LIN {X 0,Y 550.648,Z 313.22,A -85,B 0,C 180,E1 24792.082,E2 24792.082} C_VEL
LIN {X 0,Y 552.043,Z 326.315,A -85,B 0,C 180,E1 24791.727,E2 24791.727} C_VEL
LIN {X 0,Y 549.652,Z 537.017,A -85,B 0,C 180,E1 24788.42,E2 24788.42} C_VEL
LIN {X 0,Y 548.241,Z 663.349,A -85,B 0,C 180,E1 24786.457,E2 24786.457} C_VEL
LIN {X 0,Y 547.562,Z 686.68,A -85,B 0,C 180,E1 24785.907,E2 24785.907} C_VEL
LIN {X 0,Y 546.782,Z 708.656,A -85,B 0,C 180,E1 24785.202,E2 24785.202} C_VEL
LIN {X 0,Y 545.867,Z 729.431,A -85,B 0,C 180,E1 24784.342,E2 24784.342} C_VEL
LIN {X 0,Y 544.921,Z 748.48,A -85,B 0,C 180,E1 24783.397,E2 24783.397} C_VEL
LIN {X 0,Y 543.718,Z 770.272,A -85,B 0,C 180,E1 24782.102,E2 24782.102} C_VEL
LIN {X 0,Y 542.584,Z 790.428,A -85,B 0,C 180,E1 24780.692,E2 24780.692} C_VEL
LIN {X 0,Y 541.408,Z 809.495,A -85,B 0,C 180,E1 24779.129,E2 24779.129} C_VEL
LIN {X 0,Y 540.292,Z 828.469,A -85,B 0,C 180,E1 24777.342,E2 24777.342} C_VEL
LIN {X 0,Y 539.325,Z 845.154,A -85,B 0,C 180,E1 24775.532,E2 24775.532} C_VEL
LIN {X 0,Y 538.4,Z 861.896,A -85,B 0,C 180,E1 24773.451,E2 24773.451} C_VEL
LIN {X 0,Y 537.665,Z 876.959,A -85,B 0,C 180,E1 24771.303,E2 24771.303} C_VEL
LIN {X 0,Y 537.082,Z 890.104,A -85,B 0,C 180,E1 24769.125,E2 24769.125} C_VEL
LIN {X 0,Y 536.604,Z 902.808,A -85,B 0,C 180,E1 24766.674,E2 24766.674} C_VEL
LIN {X 0,Y 536.312,Z 912.539,A -85,B 0,C 180,E1 24764.465,E2 24764.465} C_VEL
LIN {X 0,Y 536.1,Z 921.347,A -85,B 0,C 180,E1 24762.056,E2 24762.056} C_VEL
LIN {X 0,Y 535.986,Z 928.174,A -85,B 0,C 180,E1 24759.772,E2 24759.772} C_VEL
LIN {X 0,Y 535.942,Z 933.843,A -85,B 0,C 180,E1 24757.287,E2 24757.287} C_VEL
LIN {X 0,Y 535.912,Z 937.597,A -85,B 0,C 180,E1 24755.029,E2 24755.029} C_VEL
LIN {X 0,Y 535.912,Z 940.056,A -85,B 0,C 180,E1 24752.565,E2 24752.565} C_VEL
LIN {X 0,Y 535.899,Z 940.94,A -85,B 0,C 180,E1 24750.32,E2 24750.32} C_VEL
LIN {X 0,Y 535.909,Z 940.323,A -85,B 0,C 180,E1 24747.86,E2 24747.86} C_VEL
LIN {X 0,Y 535.908,Z 938.502,A -85,B 0,C 180,E1 24745.719,E2 24745.719} C_VEL
LIN {X 0,Y 535.929,Z 934.666,A -85,B 0,C 180,E1 24743.141,E2 24743.141} C_VEL
LIN {X 0,Y 535.971,Z 930.06,A -85,B 0,C 180,E1 24740.983,E2 24740.983} C_VEL
LIN {X 0,Y 536.079,Z 923.115,A -85,B 0,C 180,E1 24738.487,E2 24738.487} C_VEL
LIN {X 0,Y 536.247,Z 915.403,A -85,B 0,C 180,E1 24736.271,E2 24736.271} C_VEL
LIN {X 0,Y 536.536,Z 904.879,A -85,B 0,C 180,E1 24733.767,E2 24733.767} C_VEL
LIN {X 0,Y 536.925,Z 893.82,A -85,B 0,C 180,E1 24731.543,E2 24731.543} C_VEL
LIN {X 0,Y 537.476,Z 880.753,A -85,B 0,C 180,E1 24729.3,E2 24729.3} C_VEL
LIN {X 0,Y 538.196,Z 866.294,A -85,B 0,C 180,E1 24727.141,E2 24727.141} C_VEL
LIN {X 0,Y 538.959,Z 851.402,A -85,B 0,C 180,E1 24725.211,E2 24725.211} C_VEL
LIN {X 0,Y 539.998,Z 833.11,A -85,B 0,C 180,E1 24723.141,E2 24723.141} C_VEL
LIN {X 0,Y 541.108,Z 815.109,A -85,B 0,C 180,E1 24721.366,E2 24721.366} C_VEL
LIN {X 0,Y 542.234,Z 795.587,A -85,B 0,C 180,E1 24719.713,E2 24719.713} C_VEL
LIN {X 0,Y 543.467,Z 774.991,A -85,B 0,C 180,E1 24718.209,E2 24718.209} C_VEL
LIN {X 0,Y 544.518,Z 755.81,A -85,B 0,C 180,E1 24717.013,E2 24717.013} C_VEL
LIN {X 0,Y 545.684,Z 733.227,A -85,B 0,C 180,E1 24715.833,E2 24715.833} C_VEL
LIN {X 0,Y 546.564,Z 713.963,A -85,B 0,C 180,E1 24715.004,E2 24715.004} C_VEL
LIN {X 0,Y 547.426,Z 690.328,A -85,B 0,C 180,E1 24714.196,E2 24714.196} C_VEL
LIN {X 0,Y 548.102,Z 668.726,A -85,B 0,C 180,E1 24713.65,E2 24713.65} C_VEL
LIN {X 0,Y 548.612,Z 636.425,A -85,B 0,C 180,E1 24713.105,E2 24713.105} C_VEL
LIN {X 0,Y 550.837,Z 428.699,A -85,B 0,C 180,E1 24709.893,E2 24709.893} C_VEL
LIN {X 0,Y 551.901,Z 323.442,A -85,B 0,C 180,E1 24708.21,E2 24708.21} C_VEL
LIN {X 0,Y 550.534,Z 311.332,A -85,B 0,C 180,E1 24707.849,E2 24707.849} C_VEL
LIN {X 0,Y 551.844,Z 265.411,A -85,B 0,C 180,E1 24705.585,E2 24705.585} C_VEL
LIN {X 0,Y 551.838,Z 260.378,A -85,B 0,C 180,E1 24705.331,E2 24705.331} C_VEL
LIN {X 0,Y 538.877,Z 237.428,A -85,B 0,C 180,E1 24702.918,E2 24702.918} C_VEL
LIN {X 0,Y 536.568,Z 233.016,A -85,B 0,C 180,E1 24702.42,E2 24702.42} C_VEL
LIN {X 0,Y 536.404,Z 232.242,A -85,B 0,C 180,E1 24702.2,E2 24702.2} C_VEL
LIN {X 0,Y 536.397,Z 232.226,A -85,B 0,C 180,E1 24699.191,E2 24699.191} C_VEL
LIN {X 0,Y 536.392,Z 232.232,A -85,B 0,C 180,E1 24695.819,E2 24695.819} C_VEL
LIN {X 0,Y 536.45,Z 232.224,A -85,B 0,C 180,E1 24692.592,E2 24692.592} C_VEL
LIN {X 0,Y 536.392,Z 232.227,A -85,B 0,C 180,E1 24689.357,E2 24689.357} C_VEL
LIN {X 0,Y 536.439,Z 232.22,A -85,B 0,C 180,E1 24686.052,E2 24686.052} C_VEL
LIN {X 0,Y 536.408,Z 232.228,A -85,B 0,C 180,E1 24682.928,E2 24682.928} C_VEL
LIN {X 0,Y 536.41,Z 232.224,A -85,B 0,C 180,E1 24679.491,E2 24679.491} C_VEL
LIN {X 0,Y 536.461,Z 232.226,A -85,B 0,C 180,E1 24676.235,E2 24676.235} C_VEL
LIN {X 0,Y 536.408,Z 232.226,A -85,B 0,C 180,E1 24672.925,E2 24672.925} C_VEL
LIN {X 0,Y 536.44,Z 232.221,A -85,B 0,C 180,E1 24669.549,E2 24669.549} C_VEL
LIN {X 0,Y 536.44,Z 232.223,A -85,B 0,C 180,E1 24666.314,E2 24666.314} C_VEL
LIN {X 0,Y 536.419,Z 232.224,A -85,B 0,C 180,E1 24662.992,E2 24662.992} C_VEL
LIN {X 0,Y 536.468,Z 232.223,A -85,B 0,C 180,E1 24659.68,E2 24659.68} C_VEL
LIN {X 0,Y 536.429,Z 232.221,A -85,B 0,C 180,E1 24656.367,E2 24656.367} C_VEL
LIN {X 0,Y 536.434,Z 232.221,A -85,B 0,C 180,E1 24652.934,E2 24652.934} C_VEL
LIN {X 0,Y 536.464,Z 232.224,A -85,B 0,C 180,E1 24649.585,E2 24649.585} C_VEL
LIN {X 0,Y 536.435,Z 232.22,A -85,B 0,C 180,E1 24646.191,E2 24646.191} C_VEL
LIN {X 0,Y 536.446,Z 232.22,A -85,B 0,C 180,E1 24642.762,E2 24642.762} C_VEL
LIN {X 0,Y 536.462,Z 232.223,A -85,B 0,C 180,E1 24639.331,E2 24639.331} C_VEL
LIN {X 0,Y 536.442,Z 232.221,A -85,B 0,C 180,E1 24635.966,E2 24635.966} C_VEL
LIN {X 0,Y 536.448,Z 232.221,A -85,B 0,C 180,E1 24632.469,E2 24632.469} C_VEL
LIN {X 0,Y 536.458,Z 232.224,A -85,B 0,C 180,E1 24629.15,E2 24629.15} C_VEL
LIN {X 0,Y 536.448,Z 232.221,A -85,B 0,C 180,E1 24625.745,E2 24625.745} C_VEL
LIN {X 0,Y 536.459,Z 232.218,A -85,B 0,C 180,E1 24625.468,E2 24625.468} C_VEL
LIN {X 0,Y 535.474,Z 232.341,A -85,B 0,C 180,E1 24624.645,E2 24624.645} C_VEL
LIN {X 0,Y 529.028,Z 233.146,A -85,B 0,C 180,E1 24622.334,E2 24622.334} C_VEL
LIN {X 0,Y 528.509,Z 233.214,A -85,B 0,C 180,E1 24621.732,E2 24621.732} C_VEL
LIN {X 0,Y 528.521,Z 233.209,A -85,B 0,C 180,E1 24618.192,E2 24618.192} C_VEL
LIN {X 0,Y 528.511,Z 233.211,A -85,B 0,C 180,E1 24614.731,E2 24614.731} C_VEL
LIN {X 0,Y 528.521,Z 233.206,A -85,B 0,C 180,E1 24611.319,E2 24611.319} C_VEL
LIN {X 0,Y 528.518,Z 233.207,A -85,B 0,C 180,E1 24607.804,E2 24607.804} C_VEL
LIN {X 0,Y 528.507,Z 233.209,A -85,B 0,C 180,E1 24604.428,E2 24604.428} C_VEL
LIN {X 0,Y 528.524,Z 233.213,A -85,B 0,C 180,E1 24600.969,E2 24600.969} C_VEL
LIN {X 0,Y 528.522,Z 233.212,A -85,B 0,C 180,E1 24597.472,E2 24597.472} C_VEL
LIN {X 0,Y 528.501,Z 233.211,A -85,B 0,C 180,E1 24594.121,E2 24594.121} C_VEL
LIN {X 0,Y 528.506,Z 233.193,A -85,B 0,C 180,E1 24590.604,E2 24590.604} C_VEL
LIN {X 0,Y 528.52,Z 233.186,A -85,B 0,C 180,E1 24587.166,E2 24587.166} C_VEL
LIN {X 0,Y 528.496,Z 233.207,A -85,B 0,C 180,E1 24583.792,E2 24583.792} C_VEL
LIN {X 0,Y 528.557,Z 233.488,A -85,B 0,C 180,E1 24582.621,E2 24582.621} C_VEL
LIN {X 0,Y 529.881,Z 236.792,A -85,B 0,C 180,E1 24582.198,E2 24582.198} C_VEL
LIN {X 0,Y 538.085,Z 254.046,A -85,B 0,C 180,E1 24580.223,E2 24580.223} C_VEL
LIN {X 0,Y 540.404,Z 259.527,A -85,B 0,C 180,E1 24579.64,E2 24579.64} C_VEL
LIN {X 0,Y 538.059,Z 312.95,A -85,B 0,C 180,E1 24576.242,E2 24576.242} C_VEL
LIN {X 0,Y 535.935,Z 366.94,A -85,B 0,C 180,E1 24572.888,E2 24572.888} C_VEL
LIN {X 0,Y 534.408,Z 415.343,A -85,B 0,C 180,E1 24569.964,E2 24569.964} C_VEL
LIN {X 0,Y 535.85,Z 428.483,A -85,B 0,C 180,E1 24569.659,E2 24569.659} C_VEL
LIN {X 0,Y 533.728,Z 628.852,A -85,B 0,C 180,E1 24566.685,E2 24566.685} C_VEL
LIN {X 0,Y 533.273,Z 647.783,A -85,B 0,C 180,E1 24566.202,E2 24566.202} C_VEL
LIN {X 0,Y 532.702,Z 665.893,A -85,B 0,C 180,E1 24565.534,E2 24565.534} C_VEL
LIN {X 0,Y 532.056,Z 682.703,A -85,B 0,C 180,E1 24564.718,E2 24564.718} C_VEL
LIN {X 0,Y 531.31,Z 699.567,A -85,B 0,C 180,E1 24563.681,E2 24563.681} C_VEL
LIN {X 0,Y 530.562,Z 715.414,A -85,B 0,C 180,E1 24562.475,E2 24562.475} C_VEL
LIN {X 0,Y 529.834,Z 730.891,A -85,B 0,C 180,E1 24561.045,E2 24561.045} C_VEL
LIN {X 0,Y 529.242,Z 745.559,A -85,B 0,C 180,E1 24559.442,E2 24559.442} C_VEL
LIN {X 0,Y 528.785,Z 758.201,A -85,B 0,C 180,E1 24557.775,E2 24557.775} C_VEL
LIN {X 0,Y 528.433,Z 769.398,A -85,B 0,C 180,E1 24555.985,E2 24555.985} C_VEL
LIN {X 0,Y 528.19,Z 778.61,A -85,B 0,C 180,E1 24554.183,E2 24554.183} C_VEL
LIN {X 0,Y 528.035,Z 786.5,A -85,B 0,C 180,E1 24552.252,E2 24552.252} C_VEL
LIN {X 0,Y 527.956,Z 792.73,A -85,B 0,C 180,E1 24550.257,E2 24550.257} C_VEL
LIN {X 0,Y 527.921,Z 797.031,A -85,B 0,C 180,E1 24548.328,E2 24548.328} C_VEL
LIN {X 0,Y 527.915,Z 799.808,A -85,B 0,C 180,E1 24546.328,E2 24546.328} C_VEL
LIN {X 0,Y 527.912,Z 800.934,A -85,B 0,C 180,E1 24544.298,E2 24544.298} C_VEL
LIN {X 0,Y 527.911,Z 800.355,A -85,B 0,C 180,E1 24542.232,E2 24542.232} C_VEL
LIN {X 0,Y 527.918,Z 798.144,A -85,B 0,C 180,E1 24540.252,E2 24540.252} C_VEL
LIN {X 0,Y 527.94,Z 794.185,A -85,B 0,C 180,E1 24538.232,E2 24538.232} C_VEL
LIN {X 0,Y 528.006,Z 788.481,A -85,B 0,C 180,E1 24536.232,E2 24536.232} C_VEL
LIN {X 0,Y 528.134,Z 781.189,A -85,B 0,C 180,E1 24534.308,E2 24534.308} C_VEL
LIN {X 0,Y 528.35,Z 772.33,A -85,B 0,C 180,E1 24532.458,E2 24532.458} C_VEL
LIN {X 0,Y 528.666,Z 761.804,A -85,B 0,C 180,E1 24530.671,E2 24530.671} C_VEL
LIN {X 0,Y 529.079,Z 750.063,A -85,B 0,C 180,E1 24529.024,E2 24529.024} C_VEL
LIN {X 0,Y 529.597,Z 736.845,A -85,B 0,C 180,E1 24527.479,E2 24527.479} C_VEL
LIN {X 0,Y 530.349,Z 720.375,A -85,B 0,C 180,E1 24525.854,E2 24525.854} C_VEL
LIN {X 0,Y 531.128,Z 704.59,A -85,B 0,C 180,E1 24524.569,E2 24524.569} C_VEL
LIN {X 0,Y 531.862,Z 689.465,A -85,B 0,C 180,E1 24523.558,E2 24523.558} C_VEL
LIN {X 0,Y 532.593,Z 671.915,A -85,B 0,C 180,E1 24522.618,E2 24522.618} C_VEL
LIN {X 0,Y 533.228,Z 653.953,A -85,B 0,C 180,E1 24521.88,E2 24521.88} C_VEL
LIN {X 0,Y 533.755,Z 635.41,A -85,B 0,C 180,E1 24521.334,E2 24521.334} C_VEL
LIN {X 0,Y 534.126,Z 614.34,A -85,B 0,C 180,E1 24520.945,E2 24520.945} C_VEL
LIN {X 0,Y 536.283,Z 425.675,A -85,B 0,C 180,E1 24518.106,E2 24518.106} C_VEL
LIN {X 0,Y 534.682,Z 413.113,A -85,B 0,C 180,E1 24517.757,E2 24517.757} C_VEL
LIN {X 0,Y 536.913,Z 356.868,A -85,B 0,C 180,E1 24514.285,E2 24514.285} C_VEL
LIN {X 0,Y 539.366,Z 302.398,A -85,B 0,C 180,E1 24510.84,E2 24510.84} C_VEL
LIN {X 0,Y 541.512,Z 260.702,A -85,B 0,C 180,E1 24508.148,E2 24508.148} C_VEL
LIN {X 0,Y 532.642,Z 242.077,A -85,B 0,C 180,E1 24505.936,E2 24505.936} C_VEL
LIN {X 0,Y 528.566,Z 233.729,A -85,B 0,C 180,E1 24504.86,E2 24504.86} C_VEL
LIN {X 0,Y 528.459,Z 233.211,A -85,B 0,C 180,E1 24504.597,E2 24504.597} C_VEL
LIN {X 0,Y 528.475,Z 233.203,A -85,B 0,C 180,E1 24501.437,E2 24501.437} C_VEL
LIN {X 0,Y 528.442,Z 233.221,A -85,B 0,C 180,E1 24498.077,E2 24498.077} C_VEL
LIN {X 0,Y 528.511,Z 233.213,A -85,B 0,C 180,E1 24494.797,E2 24494.797} C_VEL
LIN {X 0,Y 528.445,Z 233.219,A -85,B 0,C 180,E1 24491.569,E2 24491.569} C_VEL
LIN {X 0,Y 528.45,Z 233.215,A -85,B 0,C 180,E1 24488.048,E2 24488.048} C_VEL
LIN {X 0,Y 528.484,Z 233.215,A -85,B 0,C 180,E1 24484.883,E2 24484.883} C_VEL
LIN {X 0,Y 528.44,Z 233.219,A -85,B 0,C 180,E1 24481.626,E2 24481.626} C_VEL
LIN {X 0,Y 528.508,Z 233.218,A -85,B 0,C 180,E1 24478.373,E2 24478.373} C_VEL
LIN {X 0,Y 528.442,Z 233.22,A -85,B 0,C 180,E1 24475.115,E2 24475.115} C_VEL
LIN {X 0,Y 528.449,Z 233.216,A -85,B 0,C 180,E1 24471.623,E2 24471.623} C_VEL
LIN {X 0,Y 528.484,Z 233.218,A -85,B 0,C 180,E1 24468.431,E2 24468.431} C_VEL
LIN {X 0,Y 528.437,Z 233.215,A -85,B 0,C 180,E1 24465.2,E2 24465.2} C_VEL
LIN {X 0,Y 528.505,Z 233.213,A -85,B 0,C 180,E1 24461.925,E2 24461.925} C_VEL
LIN {X 0,Y 528.442,Z 233.217,A -85,B 0,C 180,E1 24458.698,E2 24458.698} C_VEL
LIN {X 0,Y 528.455,Z 233.219,A -85,B 0,C 180,E1 24455.251,E2 24455.251} C_VEL
LIN {X 0,Y 528.477,Z 233.218,A -85,B 0,C 180,E1 24452.069,E2 24452.069} C_VEL
LIN {X 0,Y 528.441,Z 233.221,A -85,B 0,C 180,E1 24448.773,E2 24448.773} C_VEL
LIN {X 0,Y 528.504,Z 233.215,A -85,B 0,C 180,E1 24445.551,E2 24445.551} C_VEL
LIN {X 0,Y 528.445,Z 233.224,A -85,B 0,C 180,E1 24442.266,E2 24442.266} C_VEL
LIN {X 0,Y 528.456,Z 233.208,A -85,B 0,C 180,E1 24438.82,E2 24438.82} C_VEL
LIN {X 0,Y 528.488,Z 233.533,A -85,B 0,C 180,E1 24438.281,E2 24438.281} C_VEL
LIN {X 0,Y 529.181,Z 235.703,A -85,B 0,C 180,E1 24438.021,E2 24438.021} C_VEL
LIN {X 0,Y 531.188,Z 239.035,A -85,B 0,C 180,E1 24437.634,E2 24437.634} C_VEL
LIN {X 0,Y 545.363,Z 264.536,A -85,B 0,C 180,E1 24434.99,E2 24434.99} C_VEL
LIN {X 0,Y 544.522,Z 313.223,A -85,B 0,C 180,E1 24432.667,E2 24432.667} C_VEL
LIN {X 0,Y 546.055,Z 327.732,A -85,B 0,C 180,E1 24432.266,E2 24432.266} C_VEL
LIN {X 0,Y 543.372,Z 538.137,A -85,B 0,C 180,E1 24428.928,E2 24428.928} C_VEL
LIN {X 0,Y 541.8,Z 663.427,A -85,B 0,C 180,E1 24426.961,E2 24426.961} C_VEL
LIN {X 0,Y 541.062,Z 686.547,A -85,B 0,C 180,E1 24426.411,E2 24426.411} C_VEL
LIN {X 0,Y 540.185,Z 708.26,A -85,B 0,C 180,E1 24425.713,E2 24425.713} C_VEL
LIN {X 0,Y 539.157,Z 729.428,A -85,B 0,C 180,E1 24424.831,E2 24424.831} C_VEL
LIN {X 0,Y 538.07,Z 749.226,A -85,B 0,C 180,E1 24423.837,E2 24423.837} C_VEL
LIN {X 0,Y 536.752,Z 770.268,A -85,B 0,C 180,E1 24422.569,E2 24422.569} C_VEL
LIN {X 0,Y 535.488,Z 790.431,A -85,B 0,C 180,E1 24421.144,E2 24421.144} C_VEL
LIN {X 0,Y 534.108,Z 810.292,A -85,B 0,C 180,E1 24419.493,E2 24419.493} C_VEL
LIN {X 0,Y 532.812,Z 829.805,A -85,B 0,C 180,E1 24417.612,E2 24417.612} C_VEL
LIN {X 0,Y 531.724,Z 846.674,A -85,B 0,C 180,E1 24415.744,E2 24415.744} C_VEL
LIN {X 0,Y 530.695,Z 863.005,A -85,B 0,C 180,E1 24413.658,E2 24413.658} C_VEL
LIN {X 0,Y 529.868,Z 877.935,A -85,B 0,C 180,E1 24411.472,E2 24411.472} C_VEL
LIN {X 0,Y 529.229,Z 890.737,A -85,B 0,C 180,E1 24409.305,E2 24409.305} C_VEL
LIN {X 0,Y 528.7,Z 903.054,A -85,B 0,C 180,E1 24406.878,E2 24406.878} C_VEL
LIN {X 0,Y 528.364,Z 912.996,A -85,B 0,C 180,E1 24404.576,E2 24404.576} C_VEL
LIN {X 0,Y 528.123,Z 921.704,A -85,B 0,C 180,E1 24402.13,E2 24402.13} C_VEL
LIN {X 0,Y 527.995,Z 928.777,A -85,B 0,C 180,E1 24399.702,E2 24399.702} C_VEL
LIN {X 0,Y 527.944,Z 934.05,A -85,B 0,C 180,E1 24397.289,E2 24397.289} C_VEL
LIN {X 0,Y 527.909,Z 937.915,A -85,B 0,C 180,E1 24394.888,E2 24394.888} C_VEL
LIN {X 0,Y 527.909,Z 940.124,A -85,B 0,C 180,E1 24392.496,E2 24392.496} C_VEL
LIN {X 0,Y 527.91,Z 940.984,A -85,B 0,C 180,E1 24390.107,E2 24390.107} C_VEL
LIN {X 0,Y 527.906,Z 940.189,A -85,B 0,C 180,E1 24387.611,E2 24387.611} C_VEL
LIN {X 0,Y 527.905,Z 938.047,A -85,B 0,C 180,E1 24385.219,E2 24385.219} C_VEL
LIN {X 0,Y 527.94,Z 934.253,A -85,B 0,C 180,E1 24382.818,E2 24382.818} C_VEL
LIN {X 0,Y 527.995,Z 929.039,A -85,B 0,C 180,E1 24380.406,E2 24380.406} C_VEL
LIN {X 0,Y 528.117,Z 922.052,A -85,B 0,C 180,E1 24377.979,E2 24377.979} C_VEL
LIN {X 0,Y 528.34,Z 913.883,A -85,B 0,C 180,E1 24375.645,E2 24375.645} C_VEL
LIN {X 0,Y 528.671,Z 903.843,A -85,B 0,C 180,E1 24373.292,E2 24373.292} C_VEL
LIN {X 0,Y 529.174,Z 891.995,A -85,B 0,C 180,E1 24370.92,E2 24370.92} C_VEL
LIN {X 0,Y 529.778,Z 879.337,A -85,B 0,C 180,E1 24368.754,E2 24368.754} C_VEL
LIN {X 0,Y 530.649,Z 863.832,A -85,B 0,C 180,E1 24366.455,E2 24366.455} C_VEL
LIN {X 0,Y 531.675,Z 847.665,A -85,B 0,C 180,E1 24364.371,E2 24364.371} C_VEL
LIN {X 0,Y 532.77,Z 830.337,A -85,B 0,C 180,E1 24362.443,E2 24362.443} C_VEL
LIN {X 0,Y 534.07,Z 810.922,A -85,B 0,C 180,E1 24360.564,E2 24360.564} C_VEL
LIN {X 0,Y 535.44,Z 791.173,A -85,B 0,C 180,E1 24358.913,E2 24358.913} C_VEL
LIN {X 0,Y 536.699,Z 771.131,A -85,B 0,C 180,E1 24357.488,E2 24357.488} C_VEL
LIN {X 0,Y 538.031,Z 749.95,A -85,B 0,C 180,E1 24356.202,E2 24356.202} C_VEL
LIN {X 0,Y 539.095,Z 730.661,A -85,B 0,C 180,E1 24355.227,E2 24355.227} C_VEL
LIN {X 0,Y 540.164,Z 709.052,A -85,B 0,C 180,E1 24354.316,E2 24354.316} C_VEL
LIN {X 0,Y 541.044,Z 686.986,A -85,B 0,C 180,E1 24353.601,E2 24353.601} C_VEL
LIN {X 0,Y 541.794,Z 663.936,A -85,B 0,C 180,E1 24353.049,E2 24353.049} C_VEL
LIN {X 0,Y 542.967,Z 571.712,A -85,B 0,C 180,E1 24351.595,E2 24351.595} C_VEL
LIN {X 0,Y 545.583,Z 363.045,A -85,B 0,C 180,E1 24348.302,E2 24348.302} C_VEL
LIN {X 0,Y 545.906,Z 324.77,A -85,B 0,C 180,E1 24347.669,E2 24347.669} C_VEL
LIN {X 0,Y 544.414,Z 311.611,A -85,B 0,C 180,E1 24347.276,E2 24347.276} C_VEL
LIN {X 0,Y 545.424,Z 264.362,A -85,B 0,C 180,E1 24344.966,E2 24344.966} C_VEL
LIN {X 0,Y 530.735,Z 237.869,A -85,B 0,C 180,E1 24342.119,E2 24342.119} C_VEL
LIN {X 0,Y 528.772,Z 234.692,A -85,B 0,C 180,E1 24341.728,E2 24341.728} C_VEL
LIN {X 0,Y 528.453,Z 233.284,A -85,B 0,C 180,E1 24341.485,E2 24341.485} C_VEL
LIN {X 0,Y 528.466,Z 233.219,A -85,B 0,C 180,E1 24338.082,E2 24338.082} C_VEL
LIN {X 0,Y 528.485,Z 233.213,A -85,B 0,C 180,E1 24334.845,E2 24334.845} C_VEL
LIN {X 0,Y 528.451,Z 233.214,A -85,B 0,C 180,E1 24331.481,E2 24331.481} C_VEL
LIN {X 0,Y 528.513,Z 233.212,A -85,B 0,C 180,E1 24328.227,E2 24328.227} C_VEL
LIN {X 0,Y 528.468,Z 233.212,A -85,B 0,C 180,E1 24324.956,E2 24324.956} C_VEL
LIN {X 0,Y 528.469,Z 233.214,A -85,B 0,C 180,E1 24321.534,E2 24321.534} C_VEL
LIN {X 0,Y 528.522,Z 233.207,A -85,B 0,C 180,E1 24318.251,E2 24318.251} C_VEL
LIN {X 0,Y 528.469,Z 233.213,A -85,B 0,C 180,E1 24314.911,E2 24314.911} C_VEL
LIN {X 0,Y 528.488,Z 233.21,A -85,B 0,C 180,E1 24311.458,E2 24311.458} C_VEL
LIN {X 0,Y 528.521,Z 233.216,A -85,B 0,C 180,E1 24308.157,E2 24308.157} C_VEL
LIN {X 0,Y 528.475,Z 233.21,A -85,B 0,C 180,E1 24304.776,E2 24304.776} C_VEL
LIN {X 0,Y 528.511,Z 233.2,A -85,B 0,C 180,E1 24301.41,E2 24301.41} C_VEL
LIN {X 0,Y 528.515,Z 233.216,A -85,B 0,C 180,E1 24298.049,E2 24298.049} C_VEL
LIN {X 0,Y 528.484,Z 233.21,A -85,B 0,C 180,E1 24294.681,E2 24294.681} C_VEL
LIN {X 0,Y 528.523,Z 233.201,A -85,B 0,C 180,E1 24291.405,E2 24291.405} C_VEL
LIN {X 0,Y 528.509,Z 233.216,A -85,B 0,C 180,E1 24287.985,E2 24287.985} C_VEL
LIN {X 0,Y 528.492,Z 233.209,A -85,B 0,C 180,E1 24284.529,E2 24284.529} C_VEL
LIN {X 0,Y 528.523,Z 233.199,A -85,B 0,C 180,E1 24281.126,E2 24281.126} C_VEL
LIN {X 0,Y 528.523,Z 233.215,A -85,B 0,C 180,E1 24277.651,E2 24277.651} C_VEL
LIN {X 0,Y 528.5,Z 233.208,A -85,B 0,C 180,E1 24274.207,E2 24274.207} C_VEL
LIN {X 0,Y 528.525,Z 233.198,A -85,B 0,C 180,E1 24270.786,E2 24270.786} C_VEL
LIN {X 0,Y 528.52,Z 233.212,A -85,B 0,C 180,E1 24267.245,E2 24267.245} C_VEL
LIN {X 0,Y 528.506,Z 233.209,A -85,B 0,C 180,E1 24263.825,E2 24263.825} C_VEL
LIN {X 0,Y 528.509,Z 233.214,A -85,B 0,C 180,E1 24261.732,E2 24261.732} C_VEL
LIN {X 0,Y 527.541,Z 233.34,A -85,B 0,C 180,E1 24260.897,E2 24260.897} C_VEL
LIN {X 0,Y 521.017,Z 234.145,A -85,B 0,C 180,E1 24258.49,E2 24258.49} C_VEL
LIN {X 0,Y 520.574,Z 234.2,A -85,B 0,C 180,E1 24257.939,E2 24257.939} C_VEL
LIN {X 0,Y 520.577,Z 234.198,A -85,B 0,C 180,E1 24254.512,E2 24254.512} C_VEL
LIN {X 0,Y 520.578,Z 234.196,A -85,B 0,C 180,E1 24250.991,E2 24250.991} C_VEL
LIN {X 0,Y 520.575,Z 234.197,A -85,B 0,C 180,E1 24247.647,E2 24247.647} C_VEL
LIN {X 0,Y 520.571,Z 234.196,A -85,B 0,C 180,E1 24244.248,E2 24244.248} C_VEL
LIN {X 0,Y 520.571,Z 234.199,A -85,B 0,C 180,E1 24240.725,E2 24240.725} C_VEL
LIN {X 0,Y 520.582,Z 234.203,A -85,B 0,C 180,E1 24237.326,E2 24237.326} C_VEL
LIN {X 0,Y 520.572,Z 234.198,A -85,B 0,C 180,E1 24233.903,E2 24233.903} C_VEL
LIN {X 0,Y 520.56,Z 234.185,A -85,B 0,C 180,E1 24230.396,E2 24230.396} C_VEL
LIN {X 0,Y 520.582,Z 234.169,A -85,B 0,C 180,E1 24226.968,E2 24226.968} C_VEL
LIN {X 0,Y 520.585,Z 234.23,A -85,B 0,C 180,E1 24223.439,E2 24223.439} C_VEL
LIN {X 0,Y 520.81,Z 235.309,A -85,B 0,C 180,E1 24223.207,E2 24223.207} C_VEL
LIN {X 0,Y 529.973,Z 254.408,A -85,B 0,C 180,E1 24220.931,E2 24220.931} C_VEL
LIN {X 0,Y 533.765,Z 263.071,A -85,B 0,C 180,E1 24219.979,E2 24219.979} C_VEL
LIN {X 0,Y 531.245,Z 315.749,A -85,B 0,C 180,E1 24216.594,E2 24216.594} C_VEL
LIN {X 0,Y 528.955,Z 368.924,A -85,B 0,C 180,E1 24213.252,E2 24213.252} C_VEL
LIN {X 0,Y 527.379,Z 414.556,A -85,B 0,C 180,E1 24210.466,E2 24210.466} C_VEL
LIN {X 0,Y 529.081,Z 429.209,A -85,B 0,C 180,E1 24210.111,E2 24210.111} C_VEL
LIN {X 0,Y 526.679,Z 629.306,A -85,B 0,C 180,E1 24207.09,E2 24207.09} C_VEL
LIN {X 0,Y 526.172,Z 648.334,A -85,B 0,C 180,E1 24206.597,E2 24206.597} C_VEL
LIN {X 0,Y 525.529,Z 666.665,A -85,B 0,C 180,E1 24205.91,E2 24205.91} C_VEL
LIN {X 0,Y 524.816,Z 683.447,A -85,B 0,C 180,E1 24205.083,E2 24205.083} C_VEL
LIN {X 0,Y 523.993,Z 700.315,A -85,B 0,C 180,E1 24204.032,E2 24204.032} C_VEL
LIN {X 0,Y 523.156,Z 716.188,A -85,B 0,C 180,E1 24202.81,E2 24202.81} C_VEL
LIN {X 0,Y 522.383,Z 730.54,A -85,B 0,C 180,E1 24201.471,E2 24201.471} C_VEL
LIN {X 0,Y 521.638,Z 744.037,A -85,B 0,C 180,E1 24199.956,E2 24199.956} C_VEL
LIN {X 0,Y 521.043,Z 755.772,A -85,B 0,C 180,E1 24198.377,E2 24198.377} C_VEL
LIN {X 0,Y 520.534,Z 768.469,A -85,B 0,C 180,E1 24196.335,E2 24196.335} C_VEL
LIN {X 0,Y 520.234,Z 778.373,A -85,B 0,C 180,E1 24194.392,E2 24194.392} C_VEL
LIN {X 0,Y 520.057,Z 786.307,A -85,B 0,C 180,E1 24192.433,E2 24192.433} C_VEL
LIN {X 0,Y 519.965,Z 792.528,A -85,B 0,C 180,E1 24190.428,E2 24190.428} C_VEL
LIN {X 0,Y 519.926,Z 796.924,A -85,B 0,C 180,E1 24188.452,E2 24188.452} C_VEL
LIN {X 0,Y 519.914,Z 799.748,A -85,B 0,C 180,E1 24186.423,E2 24186.423} C_VEL
LIN {X 0,Y 519.912,Z 800.921,A -85,B 0,C 180,E1 24184.362,E2 24184.362} C_VEL
LIN {X 0,Y 519.911,Z 800.392,A -85,B 0,C 180,E1 24182.266,E2 24182.266} C_VEL
LIN {X 0,Y 519.918,Z 798.232,A -85,B 0,C 180,E1 24180.255,E2 24180.255} C_VEL
LIN {X 0,Y 519.944,Z 794.325,A -85,B 0,C 180,E1 24178.205,E2 24178.205} C_VEL
LIN {X 0,Y 520.018,Z 788.635,A -85,B 0,C 180,E1 24176.161,E2 24176.161} C_VEL
LIN {X 0,Y 520.161,Z 781.396,A -85,B 0,C 180,E1 24174.209,E2 24174.209} C_VEL
LIN {X 0,Y 520.403,Z 772.596,A -85,B 0,C 180,E1 24172.332,E2 24172.332} C_VEL
LIN {X 0,Y 520.793,Z 761.468,A -85,B 0,C 180,E1 24170.404,E2 24170.404} C_VEL
LIN {X 0,Y 521.405,Z 749.111,A -85,B 0,C 180,E1 24168.582,E2 24168.582} C_VEL
LIN {X 0,Y 522.16,Z 735.706,A -85,B 0,C 180,E1 24166.959,E2 24166.959} C_VEL
LIN {X 0,Y 522.972,Z 721.344,A -85,B 0,C 180,E1 24165.519,E2 24165.519} C_VEL
LIN {X 0,Y 523.8,Z 706.602,A -85,B 0,C 180,E1 24164.292,E2 24164.292} C_VEL
LIN {X 0,Y 524.687,Z 690.023,A -85,B 0,C 180,E1 24163.165,E2 24163.165} C_VEL
LIN {X 0,Y 525.493,Z 672.615,A -85,B 0,C 180,E1 24162.221,E2 24162.221} C_VEL
LIN {X 0,Y 526.203,Z 654.48,A -85,B 0,C 180,E1 24161.467,E2 24161.467} C_VEL
LIN {X 0,Y 526.788,Z 635.901,A -85,B 0,C 180,E1 24160.912,E2 24160.912} C_VEL
LIN {X 0,Y 527.204,Z 615.012,A -85,B 0,C 180,E1 24160.518,E2 24160.518} C_VEL
LIN {X 0,Y 529.692,Z 426.735,A -85,B 0,C 180,E1 24157.627,E2 24157.627} C_VEL
LIN {X 0,Y 527.783,Z 412.04,A -85,B 0,C 180,E1 24157.214,E2 24157.214} C_VEL
LIN {X 0,Y 530.202,Z 356.418,A -85,B 0,C 180,E1 24153.735,E2 24153.735} C_VEL
LIN {X 0,Y 532.839,Z 302.985,A -85,B 0,C 180,E1 24150.315,E2 24150.315} C_VEL
LIN {X 0,Y 534.988,Z 264.373,A -85,B 0,C 180,E1 24147.794,E2 24147.794} C_VEL
LIN {X 0,Y 526.547,Z 246.768,A -85,B 0,C 180,E1 24145.654,E2 24145.654} C_VEL
LIN {X 0,Y 522.259,Z 238.269,A -85,B 0,C 180,E1 24144.547,E2 24144.547} C_VEL
LIN {X 0,Y 520.589,Z 234.729,A -85,B 0,C 180,E1 24144.062,E2 24144.062} C_VEL
LIN {X 0,Y 520.515,Z 234.2,A -85,B 0,C 180,E1 24143.79,E2 24143.79} C_VEL
LIN {X 0,Y 520.511,Z 234.202,A -85,B 0,C 180,E1 24140.345,E2 24140.345} C_VEL
LIN {X 0,Y 520.563,Z 234.205,A -85,B 0,C 180,E1 24137.089,E2 24137.089} C_VEL
LIN {X 0,Y 520.503,Z 234.21,A -85,B 0,C 180,E1 24133.893,E2 24133.893} C_VEL
LIN {X 0,Y 520.558,Z 234.203,A -85,B 0,C 180,E1 24130.625,E2 24130.625} C_VEL
LIN {X 0,Y 520.508,Z 234.204,A -85,B 0,C 180,E1 24127.394,E2 24127.394} C_VEL
LIN {X 0,Y 520.507,Z 234.209,A -85,B 0,C 180,E1 24123.855,E2 24123.855} C_VEL
LIN {X 0,Y 520.574,Z 234.204,A -85,B 0,C 180,E1 24120.55,E2 24120.55} C_VEL
LIN {X 0,Y 520.502,Z 234.207,A -85,B 0,C 180,E1 24117.247,E2 24117.247} C_VEL
LIN {X 0,Y 520.522,Z 234.205,A -85,B 0,C 180,E1 24113.824,E2 24113.824} C_VEL
LIN {X 0,Y 520.522,Z 234.204,A -85,B 0,C 180,E1 24110.714,E2 24110.714} C_VEL
LIN {X 0,Y 520.503,Z 234.207,A -85,B 0,C 180,E1 24107.35,E2 24107.35} C_VEL
LIN {X 0,Y 520.571,Z 234.203,A -85,B 0,C 180,E1 24104.058,E2 24104.058} C_VEL
LIN {X 0,Y 520.506,Z 234.209,A -85,B 0,C 180,E1 24100.707,E2 24100.707} C_VEL
LIN {X 0,Y 520.507,Z 234.205,A -85,B 0,C 180,E1 24097.168,E2 24097.168} C_VEL
LIN {X 0,Y 520.561,Z 234.202,A -85,B 0,C 180,E1 24093.906,E2 24093.906} C_VEL
LIN {X 0,Y 520.501,Z 234.21,A -85,B 0,C 180,E1 24090.67,E2 24090.67} C_VEL
LIN {X 0,Y 520.545,Z 234.205,A -85,B 0,C 180,E1 24087.334,E2 24087.334} C_VEL
LIN {X 0,Y 520.525,Z 234.21,A -85,B 0,C 180,E1 24084,E2 24084} C_VEL
LIN {X 0,Y 520.507,Z 234.211,A -85,B 0,C 180,E1 24080.661,E2 24080.661} C_VEL
LIN {X 0,Y 520.568,Z 234.383,A -85,B 0,C 180,E1 24079.083,E2 24079.083} C_VEL
LIN {X 0,Y 521.025,Z 236.167,A -85,B 0,C 180,E1 24078.835,E2 24078.835} C_VEL
LIN {X 0,Y 523.446,Z 240.572,A -85,B 0,C 180,E1 24078.317,E2 24078.317} C_VEL
LIN {X 0,Y 527.997,Z 248.909,A -85,B 0,C 180,E1 24077.391,E2 24077.391} C_VEL
LIN {X 0,Y 538.881,Z 268.427,A -85,B 0,C 180,E1 24075.352,E2 24075.352} C_VEL
LIN {X 0,Y 537.944,Z 313.569,A -85,B 0,C 180,E1 24073.178,E2 24073.178} C_VEL
LIN {X 0,Y 539.923,Z 329.156,A -85,B 0,C 180,E1 24072.792,E2 24072.792} C_VEL
LIN {X 0,Y 537.691,Z 498.338,A -85,B 0,C 180,E1 24070.096,E2 24070.096} C_VEL
LIN {X 0,Y 535.406,Z 663.197,A -85,B 0,C 180,E1 24067.482,E2 24067.482} C_VEL
LIN {X 0,Y 534.617,Z 686.155,A -85,B 0,C 180,E1 24066.935,E2 24066.935} C_VEL
LIN {X 0,Y 533.68,Z 707.187,A -85,B 0,C 180,E1 24066.258,E2 24066.258} C_VEL
LIN {X 0,Y 532.487,Z 729.425,A -85,B 0,C 180,E1 24065.332,E2 24065.332} C_VEL
LIN {X 0,Y 531.25,Z 750.003,A -85,B 0,C 180,E1 24064.286,E2 24064.286} C_VEL
LIN {X 0,Y 529.77,Z 771.165,A -85,B 0,C 180,E1 24062.989,E2 24062.989} C_VEL
LIN {X 0,Y 528.371,Z 791.207,A -85,B 0,C 180,E1 24061.548,E2 24061.548} C_VEL
LIN {X 0,Y 526.893,Z 810.289,A -85,B 0,C 180,E1 24059.938,E2 24059.938} C_VEL
LIN {X 0,Y 525.425,Z 830.137,A -85,B 0,C 180,E1 24057.997,E2 24057.997} C_VEL
LIN {X 0,Y 524.213,Z 846.673,A -85,B 0,C 180,E1 24056.14,E2 24056.14} C_VEL
LIN {X 0,Y 523.07,Z 863.003,A -85,B 0,C 180,E1 24054.025,E2 24054.025} C_VEL
LIN {X 0,Y 522.12,Z 878.246,A -85,B 0,C 180,E1 24051.756,E2 24051.756} C_VEL
LIN {X 0,Y 521.404,Z 890.735,A -85,B 0,C 180,E1 24049.607,E2 24049.607} C_VEL
LIN {X 0,Y 520.822,Z 902.811,A -85,B 0,C 180,E1 24047.195,E2 24047.195} C_VEL
LIN {X 0,Y 520.445,Z 912.572,A -85,B 0,C 180,E1 24044.908,E2 24044.908} C_VEL
LIN {X 0,Y 520.169,Z 921.349,A -85,B 0,C 180,E1 24042.431,E2 24042.431} C_VEL
LIN {X 0,Y 520.02,Z 928.049,A -85,B 0,C 180,E1 24040.122,E2 24040.122} C_VEL
LIN {X 0,Y 519.954,Z 933.637,A -85,B 0,C 180,E1 24037.624,E2 24037.624} C_VEL
LIN {X 0,Y 519.912,Z 937.279,A -85,B 0,C 180,E1 24035.406,E2 24035.406} C_VEL
LIN {X 0,Y 519.915,Z 939.988,A -85,B 0,C 180,E1 24032.755,E2 24032.755} C_VEL
LIN {X 0,Y 519.897,Z 940.917,A -85,B 0,C 180,E1 24030.44,E2 24030.44} C_VEL
LIN {X 0,Y 519.908,Z 940.391,A -85,B 0,C 180,E1 24027.905,E2 24027.905} C_VEL
LIN {X 0,Y 519.908,Z 938.615,A -85,B 0,C 180,E1 24025.698,E2 24025.698} C_VEL
LIN {X 0,Y 519.934,Z 935.079,A -85,B 0,C 180,E1 24023.151,E2 24023.151} C_VEL
LIN {X 0,Y 519.986,Z 930.57,A -85,B 0,C 180,E1 24020.927,E2 24020.927} C_VEL
LIN {X 0,Y 520.111,Z 924.173,A -85,B 0,C 180,E1 24018.466,E2 24018.466} C_VEL
LIN {X 0,Y 520.329,Z 916.065,A -85,B 0,C 180,E1 24016.025,E2 24016.025} C_VEL
LIN {X 0,Y 520.695,Z 905.905,A -85,B 0,C 180,E1 24013.488,E2 24013.488} C_VEL
LIN {X 0,Y 521.181,Z 894.985,A -85,B 0,C 180,E1 24011.197,E2 24011.197} C_VEL
LIN {X 0,Y 521.907,Z 881.454,A -85,B 0,C 180,E1 24008.771,E2 24008.771} C_VEL
LIN {X 0,Y 522.82,Z 867.209,A -85,B 0,C 180,E1 24006.559,E2 24006.559} C_VEL
LIN {X 0,Y 523.88,Z 851.403,A -85,B 0,C 180,E1 24004.447,E2 24004.447} C_VEL
LIN {X 0,Y 525.183,Z 833.111,A -85,B 0,C 180,E1 24002.319,E2 24002.319} C_VEL
LIN {X 0,Y 526.591,Z 814.893,A -85,B 0,C 180,E1 24000.479,E2 24000.479} C_VEL
LIN {X 0,Y 527.978,Z 795.906,A -85,B 0,C 180,E1 23998.833,E2 23998.833} C_VEL
LIN {X 0,Y 529.542,Z 774.719,A -85,B 0,C 180,E1 23997.25,E2 23997.25} C_VEL
LIN {X 0,Y 530.899,Z 754.797,A -85,B 0,C 180,E1 23995.988,E2 23995.988} C_VEL
LIN {X 0,Y 532.281,Z 733.226,A -85,B 0,C 180,E1 23994.848,E2 23994.848} C_VEL
LIN {X 0,Y 533.348,Z 713.956,A -85,B 0,C 180,E1 23994.004,E2 23994.004} C_VEL
LIN {X 0,Y 534.448,Z 689.904,A -85,B 0,C 180,E1 23993.172,E2 23993.172} C_VEL
LIN {X 0,Y 535.254,Z 668.562,A -85,B 0,C 180,E1 23992.627,E2 23992.627} C_VEL
LIN {X 0,Y 535.873,Z 635.686,A -85,B 0,C 180,E1 23992.064,E2 23992.064} C_VEL
LIN {X 0,Y 538.655,Z 428.444,A -85,B 0,C 180,E1 23988.788,E2 23988.788} C_VEL
LIN {X 0,Y 539.839,Z 326.799,A -85,B 0,C 180,E1 23987.162,E2 23987.162} C_VEL
LIN {X 0,Y 537.944,Z 311.534,A -85,B 0,C 180,E1 23986.734,E2 23986.734} C_VEL
LIN {X 0,Y 539.037,Z 268.354,A -85,B 0,C 180,E1 23984.594,E2 23984.594} C_VEL
LIN {X 0,Y 524.931,Z 242.972,A -85,B 0,C 180,E1 23981.81,E2 23981.81} C_VEL
LIN {X 0,Y 522.598,Z 238.659,A -85,B 0,C 180,E1 23981.305,E2 23981.305} C_VEL
LIN {X 0,Y 520.928,Z 235.849,A -85,B 0,C 180,E1 23980.955,E2 23980.955} C_VEL
LIN {X 0,Y 520.589,Z 234.292,A -85,B 0,C 180,E1 23980.703,E2 23980.703} C_VEL
LIN {X 0,Y 520.51,Z 234.203,A -85,B 0,C 180,E1 23977.374,E2 23977.374} C_VEL
LIN {X 0,Y 520.522,Z 234.209,A -85,B 0,C 180,E1 23973.852,E2 23973.852} C_VEL
LIN {X 0,Y 520.569,Z 234.205,A -85,B 0,C 180,E1 23970.596,E2 23970.596} C_VEL
LIN {X 0,Y 520.518,Z 234.208,A -85,B 0,C 180,E1 23967.329,E2 23967.329} C_VEL
LIN {X 0,Y 520.567,Z 234.204,A -85,B 0,C 180,E1 23964.029,E2 23964.029} C_VEL
LIN {X 0,Y 520.538,Z 234.204,A -85,B 0,C 180,E1 23960.815,E2 23960.815} C_VEL
LIN {X 0,Y 520.53,Z 234.203,A -85,B 0,C 180,E1 23957.318,E2 23957.318} C_VEL
LIN {X 0,Y 520.59,Z 234.195,A -85,B 0,C 180,E1 23954.005,E2 23954.005} C_VEL
LIN {X 0,Y 520.542,Z 234.2,A -85,B 0,C 180,E1 23950.626,E2 23950.626} C_VEL
LIN {X 0,Y 520.54,Z 234.201,A -85,B 0,C 180,E1 23947.173,E2 23947.173} C_VEL
LIN {X 0,Y 520.589,Z 234.203,A -85,B 0,C 180,E1 23943.855,E2 23943.855} C_VEL
LIN {X 0,Y 520.548,Z 234.193,A -85,B 0,C 180,E1 23940.441,E2 23940.441} C_VEL
LIN {X 0,Y 520.548,Z 234.196,A -85,B 0,C 180,E1 23936.917,E2 23936.917} C_VEL
LIN {X 0,Y 520.59,Z 234.199,A -85,B 0,C 180,E1 23933.494,E2 23933.494} C_VEL
LIN {X 0,Y 520.567,Z 234.195,A -85,B 0,C 180,E1 23930.046,E2 23930.046} C_VEL
LIN {X 0,Y 520.552,Z 234.195,A -85,B 0,C 180,E1 23926.561,E2 23926.561} C_VEL
LIN {X 0,Y 520.584,Z 234.2,A -85,B 0,C 180,E1 23923.257,E2 23923.257} C_VEL
LIN {X 0,Y 520.576,Z 234.194,A -85,B 0,C 180,E1 23919.775,E2 23919.775} C_VEL
LIN {X 0,Y 520.561,Z 234.196,A -85,B 0,C 180,E1 23916.333,E2 23916.333} C_VEL
LIN {X 0,Y 520.584,Z 234.199,A -85,B 0,C 180,E1 23912.923,E2 23912.923} C_VEL
LIN {X 0,Y 520.585,Z 234.196,A -85,B 0,C 180,E1 23909.368,E2 23909.368} C_VEL
LIN {X 0,Y 520.567,Z 234.198,A -85,B 0,C 180,E1 23905.877,E2 23905.877} C_VEL
LIN {X 0,Y 520.58,Z 234.197,A -85,B 0,C 180,E1 23902.356,E2 23902.356} C_VEL
LIN {X 0,Y 520.575,Z 234.203,A -85,B 0,C 180,E1 23898.939,E2 23898.939} C_VEL
LIN {X 0,Y 520.574,Z 234.2,A -85,B 0,C 180,E1 23897.939,E2 23897.939} C_VEL
LIN {X 0,Y 519.587,Z 234.327,A -85,B 0,C 180,E1 23897.091,E2 23897.091} C_VEL
LIN {X 0,Y 513.09,Z 235.132,A -85,B 0,C 180,E1 23894.647,E2 23894.647} C_VEL
LIN {X 0,Y 512.642,Z 235.186,A -85,B 0,C 180,E1 23894.088,E2 23894.088} C_VEL
LIN {X 0,Y 512.632,Z 235.188,A -85,B 0,C 180,E1 23890.65,E2 23890.65} C_VEL
LIN {X 0,Y 512.644,Z 235.182,A -85,B 0,C 180,E1 23887.203,E2 23887.203} C_VEL
LIN {X 0,Y 512.641,Z 235.184,A -85,B 0,C 180,E1 23883.637,E2 23883.637} C_VEL
LIN {X 0,Y 512.629,Z 235.183,A -85,B 0,C 180,E1 23880.214,E2 23880.214} C_VEL
LIN {X 0,Y 512.63,Z 235.185,A -85,B 0,C 180,E1 23876.655,E2 23876.655} C_VEL
LIN {X 0,Y 512.641,Z 235.169,A -85,B 0,C 180,E1 23873.203,E2 23873.203} C_VEL
LIN {X 0,Y 512.636,Z 235.189,A -85,B 0,C 180,E1 23869.721,E2 23869.721} C_VEL
LIN {X 0,Y 512.612,Z 235.157,A -85,B 0,C 180,E1 23866.197,E2 23866.197} C_VEL
LIN {X 0,Y 512.648,Z 235.437,A -85,B 0,C 180,E1 23864.089,E2 23864.089} C_VEL
LIN {X 0,Y 514.174,Z 238.995,A -85,B 0,C 180,E1 23863.61,E2 23863.61} C_VEL
LIN {X 0,Y 522.582,Z 256.431,A -85,B 0,C 180,E1 23861.479,E2 23861.479} C_VEL
LIN {X 0,Y 527.145,Z 266.617,A -85,B 0,C 180,E1 23860.327,E2 23860.327} C_VEL
LIN {X 0,Y 524.402,Z 319.395,A -85,B 0,C 180,E1 23856.9,E2 23856.9} C_VEL
LIN {X 0,Y 521.93,Z 372.683,A -85,B 0,C 180,E1 23853.516,E2 23853.516} C_VEL
LIN {X 0,Y 520.376,Z 413.645,A -85,B 0,C 180,E1 23850.985,E2 23850.985} C_VEL
LIN {X 0,Y 522.342,Z 430.191,A -85,B 0,C 180,E1 23850.572,E2 23850.572} C_VEL
LIN {X 0,Y 519.66,Z 629.642,A -85,B 0,C 180,E1 23847.51,E2 23847.51} C_VEL
LIN {X 0,Y 519.101,Z 648.78,A -85,B 0,C 180,E1 23847.006,E2 23847.006} C_VEL
LIN {X 0,Y 518.44,Z 666.216,A -85,B 0,C 180,E1 23846.352,E2 23846.352} C_VEL
LIN {X 0,Y 517.6,Z 684.19,A -85,B 0,C 180,E1 23845.459,E2 23845.459} C_VEL
LIN {X 0,Y 516.695,Z 701.065,A -85,B 0,C 180,E1 23844.393,E2 23844.393} C_VEL
LIN {X 0,Y 515.768,Z 716.962,A -85,B 0,C 180,E1 23843.154,E2 23843.154} C_VEL
LIN {X 0,Y 514.906,Z 731.348,A -85,B 0,C 180,E1 23841.796,E2 23841.796} C_VEL
LIN {X 0,Y 514.073,Z 744.881,A -85,B 0,C 180,E1 23840.259,E2 23840.259} C_VEL
LIN {X 0,Y 513.398,Z 756.655,A -85,B 0,C 180,E1 23838.657,E2 23838.657} C_VEL
LIN {X 0,Y 512.81,Z 767.837,A -85,B 0,C 180,E1 23836.815,E2 23836.815} C_VEL
LIN {X 0,Y 512.387,Z 777.048,A -85,B 0,C 180,E1 23834.959,E2 23834.959} C_VEL
LIN {X 0,Y 512.115,Z 784.948,A -85,B 0,C 180,E1 23832.972,E2 23832.972} C_VEL
LIN {X 0,Y 511.978,Z 791.989,A -85,B 0,C 180,E1 23830.73,E2 23830.73} C_VEL
LIN {X 0,Y 511.93,Z 796.818,A -85,B 0,C 180,E1 23828.58,E2 23828.58} C_VEL
LIN {X 0,Y 511.913,Z 799.687,A -85,B 0,C 180,E1 23826.52,E2 23826.52} C_VEL
LIN {X 0,Y 511.912,Z 800.908,A -85,B 0,C 180,E1 23824.429,E2 23824.429} C_VEL
LIN {X 0,Y 511.911,Z 800.428,A -85,B 0,C 180,E1 23822.301,E2 23822.301} C_VEL
LIN {X 0,Y 511.918,Z 798.319,A -85,B 0,C 180,E1 23820.259,E2 23820.259} C_VEL
LIN {X 0,Y 511.947,Z 794.435,A -85,B 0,C 180,E1 23818.164,E2 23818.164} C_VEL
LIN {X 0,Y 512.031,Z 788.673,A -85,B 0,C 180,E1 23816.051,E2 23816.051} C_VEL
LIN {X 0,Y 512.247,Z 781.045,A -85,B 0,C 180,E1 23813.882,E2 23813.882} C_VEL
LIN {X 0,Y 512.612,Z 772.454,A -85,B 0,C 180,E1 23811.951,E2 23811.951} C_VEL
LIN {X 0,Y 513.157,Z 762.226,A -85,B 0,C 180,E1 23810.089,E2 23810.089} C_VEL
LIN {X 0,Y 513.853,Z 750.136,A -85,B 0,C 180,E1 23808.284,E2 23808.284} C_VEL
LIN {X 0,Y 514.706,Z 736.664,A -85,B 0,C 180,E1 23806.632,E2 23806.632} C_VEL
LIN {X 0,Y 515.62,Z 722.171,A -85,B 0,C 180,E1 23805.161,E2 23805.161} C_VEL
LIN {X 0,Y 516.576,Z 706.648,A -85,B 0,C 180,E1 23803.861,E2 23803.861} C_VEL
LIN {X 0,Y 517.531,Z 690.659,A -85,B 0,C 180,E1 23802.767,E2 23802.767} C_VEL
LIN {X 0,Y 518.425,Z 673.158,A -85,B 0,C 180,E1 23801.807,E2 23801.807} C_VEL
LIN {X 0,Y 519.205,Z 655.109,A -85,B 0,C 180,E1 23801.046,E2 23801.046} C_VEL
LIN {X 0,Y 519.85,Z 636.487,A -85,B 0,C 180,E1 23800.48,E2 23800.48} C_VEL
LIN {X 0,Y 520.308,Z 616.049,A -85,B 0,C 180,E1 23800.085,E2 23800.085} C_VEL
LIN {X 0,Y 523.14,Z 427.899,A -85,B 0,C 180,E1 23797.14,E2 23797.14} C_VEL
LIN {X 0,Y 520.936,Z 410.847,A -85,B 0,C 180,E1 23796.649,E2 23796.649} C_VEL
LIN {X 0,Y 523.527,Z 356.098,A -85,B 0,C 180,E1 23793.179,E2 23793.179} C_VEL
LIN {X 0,Y 526.372,Z 303.428,A -85,B 0,C 180,E1 23789.767,E2 23789.767} C_VEL
LIN {X 0,Y 528.511,Z 268.137,A -85,B 0,C 180,E1 23787.435,E2 23787.435} C_VEL
LIN {X 0,Y 520.463,Z 251.465,A -85,B 0,C 180,E1 23785.366,E2 23785.366} C_VEL
LIN {X 0,Y 516.186,Z 243.05,A -85,B 0,C 180,E1 23784.245,E2 23784.245} C_VEL
LIN {X 0,Y 514.303,Z 239.236,A -85,B 0,C 180,E1 23783.729,E2 23783.729} C_VEL
LIN {X 0,Y 512.708,Z 235.691,A -85,B 0,C 180,E1 23783.229,E2 23783.229} C_VEL
LIN {X 0,Y 512.624,Z 235.194,A -85,B 0,C 180,E1 23782.96,E2 23782.96} C_VEL
LIN {X 0,Y 512.574,Z 235.2,A -85,B 0,C 180,E1 23779.722,E2 23779.722} C_VEL
LIN {X 0,Y 512.57,Z 235.199,A -85,B 0,C 180,E1 23776.197,E2 23776.197} C_VEL
LIN {X 0,Y 512.626,Z 235.193,A -85,B 0,C 180,E1 23772.961,E2 23772.961} C_VEL
LIN {X 0,Y 512.564,Z 235.196,A -85,B 0,C 180,E1 23769.657,E2 23769.657} C_VEL
LIN {X 0,Y 512.595,Z 235.196,A -85,B 0,C 180,E1 23766.271,E2 23766.271} C_VEL
LIN {X 0,Y 512.586,Z 235.198,A -85,B 0,C 180,E1 23763.019,E2 23763.019} C_VEL
LIN {X 0,Y 512.564,Z 235.193,A -85,B 0,C 180,E1 23759.664,E2 23759.664} C_VEL
LIN {X 0,Y 512.624,Z 235.191,A -85,B 0,C 180,E1 23756.309,E2 23756.309} C_VEL
LIN {X 0,Y 512.566,Z 235.195,A -85,B 0,C 180,E1 23753.053,E2 23753.053} C_VEL
LIN {X 0,Y 512.566,Z 235.198,A -85,B 0,C 180,E1 23749.457,E2 23749.457} C_VEL
LIN {X 0,Y 512.634,Z 235.193,A -85,B 0,C 180,E1 23746.119,E2 23746.119} C_VEL
LIN {X 0,Y 512.568,Z 235.197,A -85,B 0,C 180,E1 23742.752,E2 23742.752} C_VEL
LIN {X 0,Y 512.567,Z 235.195,A -85,B 0,C 180,E1 23739.205,E2 23739.205} C_VEL
LIN {X 0,Y 512.611,Z 235.191,A -85,B 0,C 180,E1 23736.064,E2 23736.064} C_VEL
LIN {X 0,Y 512.563,Z 235.199,A -85,B 0,C 180,E1 23732.715,E2 23732.715} C_VEL
LIN {X 0,Y 512.6,Z 235.194,A -85,B 0,C 180,E1 23729.335,E2 23729.335} C_VEL
LIN {X 0,Y 512.583,Z 235.2,A -85,B 0,C 180,E1 23726.091,E2 23726.091} C_VEL
LIN {X 0,Y 512.567,Z 235.203,A -85,B 0,C 180,E1 23722.651,E2 23722.651} C_VEL
LIN {X 0,Y 512.623,Z 235.434,A -85,B 0,C 180,E1 23719.868,E2 23719.868} C_VEL
LIN {X 0,Y 513.106,Z 237.122,A -85,B 0,C 180,E1 23719.631,E2 23719.631} C_VEL
LIN {X 0,Y 515.273,Z 240.881,A -85,B 0,C 180,E1 23719.161,E2 23719.161} C_VEL
LIN {X 0,Y 524.115,Z 257.281,A -85,B 0,C 180,E1 23717.298,E2 23717.298} C_VEL
LIN {X 0,Y 532.415,Z 272.414,A -85,B 0,C 180,E1 23715.719,E2 23715.719} C_VEL
LIN {X 0,Y 531.306,Z 314.581,A -85,B 0,C 180,E1 23713.651,E2 23713.651} C_VEL
LIN {X 0,Y 533.286,Z 330.433,A -85,B 0,C 180,E1 23713.255,E2 23713.255} C_VEL
LIN {X 0,Y 532.083,Z 465.002,A -85,B 0,C 180,E1 23711.19,E2 23711.19} C_VEL
LIN {X 0,Y 529.058,Z 663.005,A -85,B 0,C 180,E1 23708.015,E2 23708.015} C_VEL
LIN {X 0,Y 528.212,Z 685.891,A -85,B 0,C 180,E1 23707.467,E2 23707.467} C_VEL
LIN {X 0,Y 527.233,Z 706.216,A -85,B 0,C 180,E1 23706.811,E2 23706.811} C_VEL
LIN {X 0,Y 525.904,Z 728.643,A -85,B 0,C 180,E1 23705.883,E2 23705.883} C_VEL
LIN {X 0,Y 524.605,Z 748.49,A -85,B 0,C 180,E1 23704.872,E2 23704.872} C_VEL
LIN {X 0,Y 522.949,Z 770.433,A -85,B 0,C 180,E1 23703.528,E2 23703.528} C_VEL
LIN {X 0,Y 521.398,Z 790.437,A -85,B 0,C 180,E1 23702.084,E2 23702.084} C_VEL
LIN {X 0,Y 519.814,Z 809.229,A -85,B 0,C 180,E1 23700.489,E2 23700.489} C_VEL
LIN {X 0,Y 518.307,Z 827.583,A -85,B 0,C 180,E1 23698.706,E2 23698.706} C_VEL
LIN {X 0,Y 516.929,Z 844.139,A -85,B 0,C 180,E1 23696.847,E2 23696.847} C_VEL
LIN {X 0,Y 515.607,Z 861.309,A -85,B 0,C 180,E1 23694.639,E2 23694.639} C_VEL
LIN {X 0,Y 514.517,Z 876.516,A -85,B 0,C 180,E1 23692.387,E2 23692.387} C_VEL
LIN {X 0,Y 513.66,Z 889.463,A -85,B 0,C 180,E1 23690.152,E2 23690.152} C_VEL
LIN {X 0,Y 512.993,Z 901.77,A -85,B 0,C 180,E1 23687.7,E2 23687.7} C_VEL
LIN {X 0,Y 512.544,Z 911.617,A -85,B 0,C 180,E1 23685.384,E2 23685.384} C_VEL
LIN {X 0,Y 512.22,Z 920.994,A -85,B 0,C 180,E1 23682.742,E2 23682.742} C_VEL
LIN {X 0,Y 512.055,Z 927.567,A -85,B 0,C 180,E1 23680.461,E2 23680.461} C_VEL
LIN {X 0,Y 511.96,Z 933.43,A -85,B 0,C 180,E1 23677.856,E2 23677.856} C_VEL
LIN {X 0,Y 511.911,Z 937.12,A -85,B 0,C 180,E1 23675.603,E2 23675.603} C_VEL
LIN {X 0,Y 511.914,Z 939.852,A -85,B 0,C 180,E1 23673.022,E2 23673.022} C_VEL
LIN {X 0,Y 511.898,Z 940.873,A -85,B 0,C 180,E1 23670.67,E2 23670.67} C_VEL
LIN {X 0,Y 511.904,Z 940.525,A -85,B 0,C 180,E1 23668.096,E2 23668.096} C_VEL
LIN {X 0,Y 511.909,Z 938.728,A -85,B 0,C 180,E1 23665.742,E2 23665.742} C_VEL
LIN {X 0,Y 511.938,Z 935.492,A -85,B 0,C 180,E1 23663.269,E2 23663.269} C_VEL
LIN {X 0,Y 512.003,Z 930.571,A -85,B 0,C 180,E1 23660.784,E2 23660.784} C_VEL
LIN {X 0,Y 512.141,Z 924.172,A -85,B 0,C 180,E1 23658.284,E2 23658.284} C_VEL
LIN {X 0,Y 512.373,Z 916.339,A -85,B 0,C 180,E1 23655.88,E2 23655.88} C_VEL
LIN {X 0,Y 512.779,Z 906.419,A -85,B 0,C 180,E1 23653.343,E2 23653.343} C_VEL
LIN {X 0,Y 513.318,Z 895.567,A -85,B 0,C 180,E1 23651.016,E2 23651.016} C_VEL
LIN {X 0,Y 514.122,Z 882.152,A -85,B 0,C 180,E1 23648.553,E2 23648.553} C_VEL
LIN {X 0,Y 515.121,Z 868.003,A -85,B 0,C 180,E1 23646.309,E2 23646.309} C_VEL
LIN {X 0,Y 516.295,Z 852.33,A -85,B 0,C 180,E1 23644.167,E2 23644.167} C_VEL
LIN {X 0,Y 517.689,Z 834.77,A -85,B 0,C 180,E1 23642.071,E2 23642.071} C_VEL
LIN {X 0,Y 519.124,Z 817.686,A -85,B 0,C 180,E1 23640.302,E2 23640.302} C_VEL
LIN {X 0,Y 520.758,Z 797.781,A -85,B 0,C 180,E1 23638.516,E2 23638.516} C_VEL
LIN {X 0,Y 522.435,Z 777.569,A -85,B 0,C 180,E1 23636.957,E2 23636.957} C_VEL
LIN {X 0,Y 523.97,Z 756.804,A -85,B 0,C 180,E1 23635.608,E2 23635.608} C_VEL
LIN {X 0,Y 525.565,Z 734.508,A -85,B 0,C 180,E1 23634.397,E2 23634.397} C_VEL
LIN {X 0,Y 526.761,Z 714.693,A -85,B 0,C 180,E1 23633.516,E2 23633.516} C_VEL
LIN {X 0,Y 527.958,Z 691.227,A -85,B 0,C 180,E1 23632.686,E2 23632.686} C_VEL
LIN {X 0,Y 528.812,Z 670.347,A -85,B 0,C 180,E1 23632.139,E2 23632.139} C_VEL
LIN {X 0,Y 529.511,Z 639.656,A -85,B 0,C 180,E1 23631.592,E2 23631.592} C_VEL
LIN {X 0,Y 532.484,Z 434.053,A -85,B 0,C 180,E1 23628.318,E2 23628.318} C_VEL
LIN {X 0,Y 533.283,Z 327.548,A -85,B 0,C 180,E1 23626.66,E2 23626.66} C_VEL
LIN {X 0,Y 531.434,Z 312.971,A -85,B 0,C 180,E1 23626.259,E2 23626.259} C_VEL
LIN {X 0,Y 532.692,Z 272.277,A -85,B 0,C 180,E1 23624.211,E2 23624.211} C_VEL
LIN {X 0,Y 519.686,Z 248.67,A -85,B 0,C 180,E1 23621.588,E2 23621.588} C_VEL
LIN {X 0,Y 515.276,Z 240.663,A -85,B 0,C 180,E1 23620.626,E2 23620.626} C_VEL
LIN {X 0,Y 512.825,Z 236.392,A -85,B 0,C 180,E1 23620.083,E2 23620.083} C_VEL
LIN {X 0,Y 512.574,Z 235.23,A -85,B 0,C 180,E1 23619.828,E2 23619.828} C_VEL
LIN {X 0,Y 512.632,Z 235.189,A -85,B 0,C 180,E1 23616.504,E2 23616.504} C_VEL
LIN {X 0,Y 512.586,Z 235.199,A -85,B 0,C 180,E1 23613.105,E2 23613.105} C_VEL
LIN {X 0,Y 512.58,Z 235.194,A -85,B 0,C 180,E1 23609.572,E2 23609.572} C_VEL
LIN {X 0,Y 512.637,Z 235.184,A -85,B 0,C 180,E1 23606.207,E2 23606.207} C_VEL
LIN {X 0,Y 512.596,Z 235.193,A -85,B 0,C 180,E1 23602.841,E2 23602.841} C_VEL
LIN {X 0,Y 512.59,Z 235.191,A -85,B 0,C 180,E1 23599.366,E2 23599.366} C_VEL
LIN {X 0,Y 512.645,Z 235.188,A -85,B 0,C 180,E1 23595.963,E2 23595.963} C_VEL
LIN {X 0,Y 512.605,Z 235.194,A -85,B 0,C 180,E1 23592.619,E2 23592.619} C_VEL
LIN {X 0,Y 512.597,Z 235.19,A -85,B 0,C 180,E1 23589.091,E2 23589.091} C_VEL
LIN {X 0,Y 512.646,Z 235.18,A -85,B 0,C 180,E1 23585.709,E2 23585.709} C_VEL
LIN {X 0,Y 512.626,Z 235.19,A -85,B 0,C 180,E1 23582.236,E2 23582.236} C_VEL
LIN {X 0,Y 512.605,Z 235.192,A -85,B 0,C 180,E1 23578.771,E2 23578.771} C_VEL
LIN {X 0,Y 512.638,Z 235.185,A -85,B 0,C 180,E1 23575.302,E2 23575.302} C_VEL
LIN {X 0,Y 512.648,Z 235.18,A -85,B 0,C 180,E1 23571.815,E2 23571.815} C_VEL
LIN {X 0,Y 512.613,Z 235.191,A -85,B 0,C 180,E1 23568.411,E2 23568.411} C_VEL
LIN {X 0,Y 512.633,Z 235.184,A -85,B 0,C 180,E1 23564.9,E2 23564.9} C_VEL
LIN {X 0,Y 512.644,Z 235.178,A -85,B 0,C 180,E1 23561.424,E2 23561.424} C_VEL
LIN {X 0,Y 512.625,Z 235.192,A -85,B 0,C 180,E1 23558.008,E2 23558.008} C_VEL
LIN {X 0,Y 512.629,Z 235.183,A -85,B 0,C 180,E1 23554.466,E2 23554.466} C_VEL
LIN {X 0,Y 512.642,Z 235.177,A -85,B 0,C 180,E1 23551.073,E2 23551.073} C_VEL
LIN {X 0,Y 512.641,Z 235.194,A -85,B 0,C 180,E1 23547.564,E2 23547.564} C_VEL
LIN {X 0,Y 512.63,Z 235.184,A -85,B 0,C 180,E1 23544.042,E2 23544.042} C_VEL
LIN {X 0,Y 512.645,Z 235.175,A -85,B 0,C 180,E1 23540.52,E2 23540.52} C_VEL
LIN {X 0,Y 512.637,Z 235.184,A -85,B 0,C 180,E1 23536.95,E2 23536.95} C_VEL
LIN {X 0,Y 512.642,Z 235.186,A -85,B 0,C 180,E1 23534.088,E2 23534.088} C_VEL
LIN {X 0,Y 511.634,Z 235.318,A -85,B 0,C 180,E1 23533.227,E2 23533.227} C_VEL
LIN {X 0,Y 505.218,Z 236.11,A -85,B 0,C 180,E1 23530.808,E2 23530.808} C_VEL
LIN {X 0,Y 504.706,Z 236.174,A -85,B 0,C 180,E1 23530.177,E2 23530.177} C_VEL
LIN {X 0,Y 504.692,Z 236.175,A -85,B 0,C 180,E1 23526.608,E2 23526.608} C_VEL
LIN {X 0,Y 504.704,Z 236.171,A -85,B 0,C 180,E1 23523.072,E2 23523.072} C_VEL
LIN {X 0,Y 504.704,Z 236.169,A -85,B 0,C 180,E1 23519.558,E2 23519.558} C_VEL
LIN {X 0,Y 504.689,Z 236.173,A -85,B 0,C 180,E1 23516.093,E2 23516.093} C_VEL
LIN {X 0,Y 504.684,Z 236.145,A -85,B 0,C 180,E1 23512.601,E2 23512.601} C_VEL
LIN {X 0,Y 504.708,Z 236.182,A -85,B 0,C 180,E1 23509.08,E2 23509.08} C_VEL
LIN {X 0,Y 504.699,Z 236.148,A -85,B 0,C 180,E1 23505.513,E2 23505.513} C_VEL
LIN {X 0,Y 504.735,Z 236.353,A -85,B 0,C 180,E1 23504.883,E2 23504.883} C_VEL
LIN {X 0,Y 506.069,Z 239.783,A -85,B 0,C 180,E1 23504.416,E2 23504.416} C_VEL
LIN {X 0,Y 511.197,Z 249.997,A -85,B 0,C 180,E1 23503.086,E2 23503.086} C_VEL
LIN {X 0,Y 519.877,Z 268.51,A -85,B 0,C 180,E1 23500.865,E2 23500.865} C_VEL
LIN {X 0,Y 520.544,Z 270.168,A -85,B 0,C 180,E1 23500.683,E2 23500.683} C_VEL
LIN {X 0,Y 517.575,Z 323.041,A -85,B 0,C 180,E1 23497.215,E2 23497.215} C_VEL
LIN {X 0,Y 514.96,Z 375.59,A -85,B 0,C 180,E1 23493.842,E2 23493.842} C_VEL
LIN {X 0,Y 513.434,Z 412.862,A -85,B 0,C 180,E1 23491.515,E2 23491.515} C_VEL
LIN {X 0,Y 515.636,Z 431.273,A -85,B 0,C 180,E1 23491.043,E2 23491.043} C_VEL
LIN {X 0,Y 512.674,Z 629.827,A -85,B 0,C 180,E1 23487.944,E2 23487.944} C_VEL
LIN {X 0,Y 512.065,Z 649.02,A -85,B 0,C 180,E1 23487.434,E2 23487.434} C_VEL
LIN {X 0,Y 511.32,Z 666.983,A -85,B 0,C 180,E1 23486.75,E2 23486.75} C_VEL
LIN {X 0,Y 510.408,Z 684.931,A -85,B 0,C 180,E1 23485.845,E2 23485.845} C_VEL
LIN {X 0,Y 509.419,Z 701.815,A -85,B 0,C 180,E1 23484.765,E2 23484.765} C_VEL
LIN {X 0,Y 508.4,Z 717.737,A -85,B 0,C 180,E1 23483.508,E2 23483.508} C_VEL
LIN {X 0,Y 507.447,Z 732.155,A -85,B 0,C 180,E1 23482.13,E2 23482.13} C_VEL
LIN {X 0,Y 506.526,Z 745.723,A -85,B 0,C 180,E1 23480.572,E2 23480.572} C_VEL
LIN {X 0,Y 505.771,Z 757.536,A -85,B 0,C 180,E1 23478.946,E2 23478.946} C_VEL
LIN {X 0,Y 505.144,Z 768.143,A -85,B 0,C 180,E1 23477.193,E2 23477.193} C_VEL
LIN {X 0,Y 504.614,Z 778.012,A -85,B 0,C 180,E1 23475.192,E2 23475.192} C_VEL
LIN {X 0,Y 504.288,Z 785.94,A -85,B 0,C 180,E1 23473.175,E2 23473.175} C_VEL
LIN {X 0,Y 504.082,Z 792.218,A -85,B 0,C 180,E1 23471.107,E2 23471.107} C_VEL
LIN {X 0,Y 503.969,Z 796.725,A -85,B 0,C 180,E1 23469.078,E2 23469.078} C_VEL
LIN {X 0,Y 503.935,Z 799.748,A -85,B 0,C 180,E1 23466.993,E2 23466.993} C_VEL
LIN {X 0,Y 503.922,Z 801.24,A -85,B 0,C 180,E1 23464.791,E2 23464.791} C_VEL
LIN {X 0,Y 503.921,Z 801.046,A -85,B 0,C 180,E1 23462.594,E2 23462.594} C_VEL
LIN {X 0,Y 503.941,Z 799.154,A -85,B 0,C 180,E1 23460.396,E2 23460.396} C_VEL
LIN {X 0,Y 504.002,Z 795.714,A -85,B 0,C 180,E1 23458.285,E2 23458.285} C_VEL
LIN {X 0,Y 504.156,Z 790.471,A -85,B 0,C 180,E1 23456.133,E2 23456.133} C_VEL
LIN {X 0,Y 504.418,Z 783.313,A -85,B 0,C 180,E1 23453.971,E2 23453.971} C_VEL
LIN {X 0,Y 504.826,Z 774.845,A -85,B 0,C 180,E1 23451.98,E2 23451.98} C_VEL
LIN {X 0,Y 505.425,Z 764.791,A -85,B 0,C 180,E1 23450.073,E2 23450.073} C_VEL
LIN {X 0,Y 506.165,Z 753.188,A -85,B 0,C 180,E1 23448.266,E2 23448.266} C_VEL
LIN {X 0,Y 507.081,Z 740.201,A -85,B 0,C 180,E1 23446.596,E2 23446.596} C_VEL
LIN {X 0,Y 508.058,Z 726.303,A -85,B 0,C 180,E1 23445.11,E2 23445.11} C_VEL
LIN {X 0,Y 509.077,Z 711.544,A -85,B 0,C 180,E1 23443.8,E2 23443.8} C_VEL
LIN {X 0,Y 510.137,Z 695.292,A -85,B 0,C 180,E1 23442.613,E2 23442.613} C_VEL
LIN {X 0,Y 511.141,Z 678.118,A -85,B 0,C 180,E1 23441.604,E2 23441.604} C_VEL
LIN {X 0,Y 512.046,Z 660.305,A -85,B 0,C 180,E1 23440.789,E2 23440.789} C_VEL
LIN {X 0,Y 512.781,Z 641.975,A -85,B 0,C 180,E1 23440.168,E2 23440.168} C_VEL
LIN {X 0,Y 513.327,Z 622.948,A -85,B 0,C 180,E1 23439.737,E2 23439.737} C_VEL
LIN {X 0,Y 516.626,Z 429.171,A -85,B 0,C 180,E1 23436.646,E2 23436.646} C_VEL
LIN {X 0,Y 514.155,Z 409.525,A -85,B 0,C 180,E1 23436.059,E2 23436.059} C_VEL
LIN {X 0,Y 517.025,Z 353.529,A -85,B 0,C 180,E1 23432.462,E2 23432.462} C_VEL
LIN {X 0,Y 520.118,Z 301.357,A -85,B 0,C 180,E1 23429.038,E2 23429.038} C_VEL
LIN {X 0,Y 521.981,Z 271.891,A -85,B 0,C 180,E1 23427.06,E2 23427.06} C_VEL
LIN {X 0,Y 514.425,Z 256.093,A -85,B 0,C 180,E1 23425.069,E2 23425.069} C_VEL
LIN {X 0,Y 508.7,Z 244.666,A -85,B 0,C 180,E1 23423.515,E2 23423.515} C_VEL
LIN {X 0,Y 506.445,Z 240.288,A -85,B 0,C 180,E1 23422.887,E2 23422.887} C_VEL
LIN {X 0,Y 504.722,Z 236.739,A -85,B 0,C 180,E1 23422.355,E2 23422.355} C_VEL
LIN {X 0,Y 504.629,Z 236.199,A -85,B 0,C 180,E1 23422.114,E2 23422.114} C_VEL
LIN {X 0,Y 504.668,Z 236.182,A -85,B 0,C 180,E1 23418.72,E2 23418.72} C_VEL
LIN {X 0,Y 504.648,Z 236.189,A -85,B 0,C 180,E1 23415.396,E2 23415.396} C_VEL
LIN {X 0,Y 504.628,Z 236.187,A -85,B 0,C 180,E1 23412.007,E2 23412.007} C_VEL
LIN {X 0,Y 504.691,Z 236.183,A -85,B 0,C 180,E1 23408.659,E2 23408.659} C_VEL
LIN {X 0,Y 504.631,Z 236.185,A -85,B 0,C 180,E1 23405.343,E2 23405.343} C_VEL
LIN {X 0,Y 504.63,Z 236.186,A -85,B 0,C 180,E1 23401.816,E2 23401.816} C_VEL
LIN {X 0,Y 504.689,Z 236.181,A -85,B 0,C 180,E1 23398.524,E2 23398.524} C_VEL
LIN {X 0,Y 504.627,Z 236.188,A -85,B 0,C 180,E1 23395.112,E2 23395.112} C_VEL
LIN {X 0,Y 504.63,Z 236.183,A -85,B 0,C 180,E1 23391.568,E2 23391.568} C_VEL
LIN {X 0,Y 504.685,Z 236.178,A -85,B 0,C 180,E1 23388.225,E2 23388.225} C_VEL
LIN {X 0,Y 504.622,Z 236.181,A -85,B 0,C 180,E1 23384.956,E2 23384.956} C_VEL
LIN {X 0,Y 504.645,Z 236.186,A -85,B 0,C 180,E1 23381.518,E2 23381.518} C_VEL
LIN {X 0,Y 504.657,Z 236.184,A -85,B 0,C 180,E1 23378.254,E2 23378.254} C_VEL
LIN {X 0,Y 504.624,Z 236.186,A -85,B 0,C 180,E1 23374.886,E2 23374.886} C_VEL
LIN {X 0,Y 504.671,Z 236.182,A -85,B 0,C 180,E1 23371.479,E2 23371.479} C_VEL
LIN {X 0,Y 504.642,Z 236.189,A -85,B 0,C 180,E1 23368.195,E2 23368.195} C_VEL
LIN {X 0,Y 504.629,Z 236.191,A -85,B 0,C 180,E1 23364.716,E2 23364.716} C_VEL
LIN {X 0,Y 504.686,Z 236.183,A -85,B 0,C 180,E1 23361.31,E2 23361.31} C_VEL
LIN {X 0,Y 504.666,Z 236.424,A -85,B 0,C 180,E1 23360.715,E2 23360.715} C_VEL
LIN {X 0,Y 505.097,Z 238.065,A -85,B 0,C 180,E1 23360.474,E2 23360.474} C_VEL
LIN {X 0,Y 507.439,Z 241.955,A -85,B 0,C 180,E1 23359.959,E2 23359.959} C_VEL
LIN {X 0,Y 516.794,Z 259.338,A -85,B 0,C 180,E1 23357.903,E2 23357.903} C_VEL
LIN {X 0,Y 525.932,Z 276.243,A -85,B 0,C 180,E1 23356.095,E2 23356.095} C_VEL
LIN {X 0,Y 524.72,Z 315.706,A -85,B 0,C 180,E1 23354.133,E2 23354.133} C_VEL
LIN {X 0,Y 526.675,Z 331.713,A -85,B 0,C 180,E1 23353.728,E2 23353.728} C_VEL
LIN {X 0,Y 524.843,Z 537.312,A -85,B 0,C 180,E1 23350.59,E2 23350.59} C_VEL
LIN {X 0,Y 522.749,Z 663.198,A -85,B 0,C 180,E1 23348.553,E2 23348.553} C_VEL
LIN {X 0,Y 521.833,Z 686.019,A -85,B 0,C 180,E1 23348.002,E2 23348.002} C_VEL
LIN {X 0,Y 520.803,Z 705.88,A -85,B 0,C 180,E1 23347.356,E2 23347.356} C_VEL
LIN {X 0,Y 519.334,Z 728.564,A -85,B 0,C 180,E1 23346.413,E2 23346.413} C_VEL
LIN {X 0,Y 517.839,Z 749.612,A -85,B 0,C 180,E1 23345.328,E2 23345.328} C_VEL
LIN {X 0,Y 516.138,Z 770.258,A -85,B 0,C 180,E1 23344.043,E2 23344.043} C_VEL
LIN {X 0,Y 514.405,Z 790.439,A -85,B 0,C 180,E1 23342.574,E2 23342.574} C_VEL
LIN {X 0,Y 512.669,Z 809.42,A -85,B 0,C 180,E1 23340.942,E2 23340.942} C_VEL
LIN {X 0,Y 510.959,Z 828.136,A -85,B 0,C 180,E1 23339.094,E2 23339.094} C_VEL
LIN {X 0,Y 509.468,Z 844.645,A -85,B 0,C 180,E1 23337.21,E2 23337.21} C_VEL
LIN {X 0,Y 508.035,Z 861.309,A -85,B 0,C 180,E1 23335.031,E2 23335.031} C_VEL
LIN {X 0,Y 506.824,Z 876.517,A -85,B 0,C 180,E1 23332.746,E2 23332.746} C_VEL
LIN {X 0,Y 505.885,Z 889.476,A -85,B 0,C 180,E1 23330.473,E2 23330.473} C_VEL
LIN {X 0,Y 505.134,Z 901.772,A -85,B 0,C 180,E1 23327.985,E2 23327.985} C_VEL
LIN {X 0,Y 504.628,Z 911.616,A -85,B 0,C 180,E1 23325.631,E2 23325.631} C_VEL
LIN {X 0,Y 504.262,Z 920.995,A -85,B 0,C 180,E1 23322.946,E2 23322.946} C_VEL
LIN {X 0,Y 504.073,Z 927.567,A -85,B 0,C 180,E1 23320.629,E2 23320.629} C_VEL
LIN {X 0,Y 503.961,Z 933.43,A -85,B 0,C 180,E1 23317.982,E2 23317.982} C_VEL
LIN {X 0,Y 503.912,Z 937.12,A -85,B 0,C 180,E1 23315.692,E2 23315.692} C_VEL
LIN {X 0,Y 503.913,Z 939.851,A -85,B 0,C 180,E1 23313.07,E2 23313.07} C_VEL
LIN {X 0,Y 503.899,Z 940.873,A -85,B 0,C 180,E1 23310.681,E2 23310.681} C_VEL
LIN {X 0,Y 503.905,Z 940.526,A -85,B 0,C 180,E1 23308.066,E2 23308.066} C_VEL
LIN {X 0,Y 503.907,Z 938.728,A -85,B 0,C 180,E1 23305.675,E2 23305.675} C_VEL
LIN {X 0,Y 503.939,Z 935.492,A -85,B 0,C 180,E1 23303.162,E2 23303.162} C_VEL
LIN {X 0,Y 504.015,Z 930.571,A -85,B 0,C 180,E1 23300.637,E2 23300.637} C_VEL
LIN {X 0,Y 504.168,Z 924.171,A -85,B 0,C 180,E1 23298.096,E2 23298.096} C_VEL
LIN {X 0,Y 504.431,Z 916.34,A -85,B 0,C 180,E1 23295.653,E2 23295.653} C_VEL
LIN {X 0,Y 504.89,Z 906.417,A -85,B 0,C 180,E1 23293.074,E2 23293.074} C_VEL
LIN {X 0,Y 505.501,Z 895.569,A -85,B 0,C 180,E1 23290.711,E2 23290.711} C_VEL
LIN {X 0,Y 506.402,Z 882.15,A -85,B 0,C 180,E1 23288.21,E2 23288.21} C_VEL
LIN {X 0,Y 507.495,Z 868.005,A -85,B 0,C 180,E1 23285.931,E2 23285.931} C_VEL
LIN {X 0,Y 508.8,Z 852.329,A -85,B 0,C 180,E1 23283.758,E2 23283.758} C_VEL
LIN {X 0,Y 510.305,Z 835.323,A -85,B 0,C 180,E1 23281.694,E2 23281.694} C_VEL
LIN {X 0,Y 511.835,Z 818.548,A -85,B 0,C 180,E1 23279.927,E2 23279.927} C_VEL
LIN {X 0,Y 513.589,Z 799.247,A -85,B 0,C 180,E1 23278.157,E2 23278.157} C_VEL
LIN {X 0,Y 515.258,Z 780.696,A -85,B 0,C 180,E1 23276.69,E2 23276.69} C_VEL
LIN {X 0,Y 516.985,Z 759.848,A -85,B 0,C 180,E1 23275.281,E2 23275.281} C_VEL
LIN {X 0,Y 518.609,Z 739.402,A -85,B 0,C 180,E1 23274.118,E2 23274.118} C_VEL
LIN {X 0,Y 520.086,Z 717.621,A -85,B 0,C 180,E1 23273.107,E2 23273.107} C_VEL
LIN {X 0,Y 521.306,Z 696.82,A -85,B 0,C 180,E1 23272.324,E2 23272.324} C_VEL
LIN {X 0,Y 522.325,Z 673.967,A -85,B 0,C 180,E1 23271.682,E2 23271.682} C_VEL
LIN {X 0,Y 523.08,Z 650.398,A -85,B 0,C 180,E1 23271.217,E2 23271.217} C_VEL
LIN {X 0,Y 525.231,Z 501.831,A -85,B 0,C 180,E1 23268.862,E2 23268.862} C_VEL
LIN {X 0,Y 526.921,Z 329.447,A -85,B 0,C 180,E1 23266.177,E2 23266.177} C_VEL
LIN {X 0,Y 524.984,Z 313.636,A -85,B 0,C 180,E1 23265.734,E2 23265.734} C_VEL
LIN {X 0,Y 526.359,Z 276.251,A -85,B 0,C 180,E1 23263.82,E2 23263.82} C_VEL
LIN {X 0,Y 513.937,Z 253.627,A -85,B 0,C 180,E1 23261.263,E2 23261.263} C_VEL
LIN {X 0,Y 508.794,Z 244.504,A -85,B 0,C 180,E1 23260.134,E2 23260.134} C_VEL
LIN {X 0,Y 507.054,Z 240.997,A -85,B 0,C 180,E1 23259.71,E2 23259.71} C_VEL
LIN {X 0,Y 505.066,Z 237.948,A -85,B 0,C 180,E1 23259.28,E2 23259.28} C_VEL
LIN {X 0,Y 504.683,Z 236.392,A -85,B 0,C 180,E1 23259.047,E2 23259.047} C_VEL
LIN {X 0,Y 504.633,Z 236.19,A -85,B 0,C 180,E1 23255.628,E2 23255.628} C_VEL
LIN {X 0,Y 504.678,Z 236.174,A -85,B 0,C 180,E1 23252.204,E2 23252.204} C_VEL
LIN {X 0,Y 504.657,Z 236.177,A -85,B 0,C 180,E1 23248.91,E2 23248.91} C_VEL
LIN {X 0,Y 504.644,Z 236.177,A -85,B 0,C 180,E1 23245.464,E2 23245.464} C_VEL
LIN {X 0,Y 504.705,Z 236.171,A -85,B 0,C 180,E1 23242.111,E2 23242.111} C_VEL
LIN {X 0,Y 504.663,Z 236.176,A -85,B 0,C 180,E1 23238.721,E2 23238.721} C_VEL
LIN {X 0,Y 504.653,Z 236.178,A -85,B 0,C 180,E1 23235.227,E2 23235.227} C_VEL
LIN {X 0,Y 504.703,Z 236.177,A -85,B 0,C 180,E1 23231.857,E2 23231.857} C_VEL
LIN {X 0,Y 504.678,Z 236.181,A -85,B 0,C 180,E1 23228.431,E2 23228.431} C_VEL
LIN {X 0,Y 504.661,Z 236.175,A -85,B 0,C 180,E1 23225.001,E2 23225.001} C_VEL
LIN {X 0,Y 504.707,Z 236.165,A -85,B 0,C 180,E1 23221.59,E2 23221.59} C_VEL
LIN {X 0,Y 504.687,Z 236.184,A -85,B 0,C 180,E1 23218.184,E2 23218.184} C_VEL
LIN {X 0,Y 504.668,Z 236.177,A -85,B 0,C 180,E1 23214.657,E2 23214.657} C_VEL
LIN {X 0,Y 504.702,Z 236.164,A -85,B 0,C 180,E1 23211.226,E2 23211.226} C_VEL
LIN {X 0,Y 504.704,Z 236.178,A -85,B 0,C 180,E1 23207.762,E2 23207.762} C_VEL
LIN {X 0,Y 504.678,Z 236.177,A -85,B 0,C 180,E1 23204.252,E2 23204.252} C_VEL
LIN {X 0,Y 504.688,Z 236.163,A -85,B 0,C 180,E1 23200.68,E2 23200.68} C_VEL
LIN {X 0,Y 504.705,Z 236.175,A -85,B 0,C 180,E1 23197.276,E2 23197.276} C_VEL
LIN {X 0,Y 504.695,Z 236.177,A -85,B 0,C 180,E1 23193.783,E2 23193.783} C_VEL
LIN {X 0,Y 504.689,Z 236.165,A -85,B 0,C 180,E1 23190.312,E2 23190.312} C_VEL
LIN {X 0,Y 504.703,Z 236.173,A -85,B 0,C 180,E1 23186.854,E2 23186.854} C_VEL
LIN {X 0,Y 504.706,Z 236.183,A -85,B 0,C 180,E1 23183.254,E2 23183.254} C_VEL
LIN {X 0,Y 504.691,Z 236.168,A -85,B 0,C 180,E1 23179.707,E2 23179.707} C_VEL
LIN {X 0,Y 504.704,Z 236.168,A -85,B 0,C 180,E1 23176.147,E2 23176.147} C_VEL
LIN {X 0,Y 504.694,Z 236.174,A -85,B 0,C 180,E1 23172.653,E2 23172.653} C_VEL
LIN {X 0,Y 504.706,Z 236.174,A -85,B 0,C 180,E1 23170.177,E2 23170.177} C_VEL
LIN {X 0,Y 503.73,Z 236.304,A -85,B 0,C 180,E1 23169.302,E2 23169.302} C_VEL
LIN {X 0,Y 497.275,Z 237.101,A -85,B 0,C 180,E1 23166.845,E2 23166.845} C_VEL
LIN {X 0,Y 496.76,Z 237.164,A -85,B 0,C 180,E1 23166.204,E2 23166.204} C_VEL
LIN {X 0,Y 496.752,Z 237.164,A -85,B 0,C 180,E1 23162.646,E2 23162.646} C_VEL
LIN {X 0,Y 496.769,Z 237.16,A -85,B 0,C 180,E1 23159.131,E2 23159.131} C_VEL
LIN {X 0,Y 496.767,Z 237.163,A -85,B 0,C 180,E1 23155.515,E2 23155.515} C_VEL
LIN {X 0,Y 496.742,Z 237.125,A -85,B 0,C 180,E1 23151.987,E2 23151.987} C_VEL
LIN {X 0,Y 496.746,Z 237.16,A -85,B 0,C 180,E1 23148.423,E2 23148.423} C_VEL
LIN {X 0,Y 496.774,Z 237.33,A -85,B 0,C 180,E1 23145.707,E2 23145.707} C_VEL
LIN {X 0,Y 498.317,Z 240.968,A -85,B 0,C 180,E1 23145.182,E2 23145.182} C_VEL
LIN {X 0,Y 506.792,Z 257.956,A -85,B 0,C 180,E1 23142.94,E2 23142.94} C_VEL
LIN {X 0,Y 513.963,Z 273.722,A -85,B 0,C 180,E1 23141.048,E2 23141.048} C_VEL
LIN {X 0,Y 510.777,Z 326.731,A -85,B 0,C 180,E1 23137.537,E2 23137.537} C_VEL
LIN {X 0,Y 507.956,Z 379.334,A -85,B 0,C 180,E1 23134.121,E2 23134.121} C_VEL
LIN {X 0,Y 506.519,Z 411.946,A -85,B 0,C 180,E1 23132.062,E2 23132.062} C_VEL
LIN {X 0,Y 508.953,Z 432.343,A -85,B 0,C 180,E1 23131.524,E2 23131.524} C_VEL
LIN {X 0,Y 505.716,Z 630.178,A -85,B 0,C 180,E1 23128.387,E2 23128.387} C_VEL
LIN {X 0,Y 505.051,Z 649.497,A -85,B 0,C 180,E1 23127.866,E2 23127.866} C_VEL
LIN {X 0,Y 504.227,Z 667.757,A -85,B 0,C 180,E1 23127.16,E2 23127.16} C_VEL
LIN {X 0,Y 503.24,Z 685.676,A -85,B 0,C 180,E1 23126.242,E2 23126.242} C_VEL
LIN {X 0,Y 502.165,Z 702.568,A -85,B 0,C 180,E1 23125.147,E2 23125.147} C_VEL
LIN {X 0,Y 501.054,Z 718.514,A -85,B 0,C 180,E1 23123.873,E2 23123.873} C_VEL
LIN {X 0,Y 500.007,Z 732.963,A -85,B 0,C 180,E1 23122.475,E2 23122.475} C_VEL
LIN {X 0,Y 498.995,Z 746.565,A -85,B 0,C 180,E1 23120.893,E2 23120.893} C_VEL
LIN {X 0,Y 498.156,Z 758.417,A -85,B 0,C 180,E1 23119.243,E2 23119.243} C_VEL
LIN {X 0,Y 497.406,Z 769.681,A -85,B 0,C 180,E1 23117.345,E2 23117.345} C_VEL
LIN {X 0,Y 496.851,Z 778.976,A -85,B 0,C 180,E1 23115.432,E2 23115.432} C_VEL
LIN {X 0,Y 496.468,Z 786.947,A -85,B 0,C 180,E1 23113.384,E2 23113.384} C_VEL
LIN {X 0,Y 496.219,Z 793.318,A -85,B 0,C 180,E1 23111.265,E2 23111.265} C_VEL
LIN {X 0,Y 496.08,Z 798.032,A -85,B 0,C 180,E1 23109.101,E2 23109.101} C_VEL
LIN {X 0,Y 496.033,Z 801.017,A -85,B 0,C 180,E1 23106.982,E2 23106.982} C_VEL
LIN {X 0,Y 496.017,Z 802.459,A -85,B 0,C 180,E1 23104.83,E2 23104.83} C_VEL
LIN {X 0,Y 496.018,Z 802.324,A -85,B 0,C 180,E1 23102.641,E2 23102.641} C_VEL
LIN {X 0,Y 496.049,Z 800.502,A -85,B 0,C 180,E1 23100.409,E2 23100.409} C_VEL
LIN {X 0,Y 496.13,Z 797.129,A -85,B 0,C 180,E1 23098.26,E2 23098.26} C_VEL
LIN {X 0,Y 496.313,Z 791.986,A -85,B 0,C 180,E1 23096.082,E2 23096.082} C_VEL
LIN {X 0,Y 496.6,Z 785.316,A -85,B 0,C 180,E1 23093.993,E2 23093.993} C_VEL
LIN {X 0,Y 497.041,Z 777.235,A -85,B 0,C 180,E1 23092.01,E2 23092.01} C_VEL
LIN {X 0,Y 497.668,Z 767.752,A -85,B 0,C 180,E1 23090.126,E2 23090.126} C_VEL
LIN {X 0,Y 498.445,Z 756.718,A -85,B 0,C 180,E1 23088.32,E2 23088.32} C_VEL
LIN {X 0,Y 499.414,Z 744.126,A -85,B 0,C 180,E1 23086.613,E2 23086.613} C_VEL
LIN {X 0,Y 500.475,Z 730.482,A -85,B 0,C 180,E1 23085.073,E2 23085.073} C_VEL
LIN {X 0,Y 501.626,Z 715.325,A -85,B 0,C 180,E1 23083.655,E2 23083.655} C_VEL
LIN {X 0,Y 502.749,Z 699.778,A -85,B 0,C 180,E1 23082.455,E2 23082.455} C_VEL
LIN {X 0,Y 503.869,Z 683.006,A -85,B 0,C 180,E1 23081.404,E2 23081.404} C_VEL
LIN {X 0,Y 504.867,Z 665.452,A -85,B 0,C 180,E1 23080.535,E2 23080.535} C_VEL
LIN {X 0,Y 505.713,Z 647.062,A -85,B 0,C 180,E1 23079.848,E2 23079.848} C_VEL
LIN {X 0,Y 506.391,Z 628.06,A -85,B 0,C 180,E1 23079.36,E2 23079.36} C_VEL
LIN {X 0,Y 510.164,Z 430.577,A -85,B 0,C 180,E1 23076.142,E2 23076.142} C_VEL
LIN {X 0,Y 507.407,Z 408.521,A -85,B 0,C 180,E1 23075.472,E2 23075.472} C_VEL
LIN {X 0,Y 510.615,Z 350.855,A -85,B 0,C 180,E1 23071.719,E2 23071.719} C_VEL
LIN {X 0,Y 514.043,Z 298.029,A -85,B 0,C 180,E1 23068.206,E2 23068.206} C_VEL
LIN {X 0,Y 515.493,Z 275.657,A -85,B 0,C 180,E1 23066.68,E2 23066.68} C_VEL
LIN {X 0,Y 507.322,Z 258.294,A -85,B 0,C 180,E1 23064.448,E2 23064.448} C_VEL
LIN {X 0,Y 500.89,Z 245.771,A -85,B 0,C 180,E1 23062.659,E2 23062.659} C_VEL
LIN {X 0,Y 498.662,Z 241.512,A -85,B 0,C 180,E1 23062.021,E2 23062.021} C_VEL
LIN {X 0,Y 496.887,Z 238.092,A -85,B 0,C 180,E1 23061.498,E2 23061.498} C_VEL
LIN {X 0,Y 496.745,Z 237.192,A -85,B 0,C 180,E1 23061.241,E2 23061.241} C_VEL
LIN {X 0,Y 496.69,Z 237.179,A -85,B 0,C 180,E1 23057.799,E2 23057.799} C_VEL
LIN {X 0,Y 496.697,Z 237.175,A -85,B 0,C 180,E1 23054.216,E2 23054.216} C_VEL
LIN {X 0,Y 496.747,Z 237.17,A -85,B 0,C 180,E1 23050.788,E2 23050.788} C_VEL
LIN {X 0,Y 496.691,Z 237.17,A -85,B 0,C 180,E1 23047.402,E2 23047.402} C_VEL
LIN {X 0,Y 496.69,Z 237.177,A -85,B 0,C 180,E1 23043.809,E2 23043.809} C_VEL
LIN {X 0,Y 496.757,Z 237.167,A -85,B 0,C 180,E1 23040.461,E2 23040.461} C_VEL
LIN {X 0,Y 496.698,Z 237.172,A -85,B 0,C 180,E1 23036.999,E2 23036.999} C_VEL
LIN {X 0,Y 496.688,Z 237.173,A -85,B 0,C 180,E1 23033.527,E2 23033.527} C_VEL
LIN {X 0,Y 496.745,Z 237.169,A -85,B 0,C 180,E1 23030.148,E2 23030.148} C_VEL
LIN {X 0,Y 496.696,Z 237.175,A -85,B 0,C 180,E1 23026.733,E2 23026.733} C_VEL
LIN {X 0,Y 496.689,Z 237.176,A -85,B 0,C 180,E1 23023.269,E2 23023.269} C_VEL
LIN {X 0,Y 496.747,Z 237.167,A -85,B 0,C 180,E1 23019.867,E2 23019.867} C_VEL
LIN {X 0,Y 496.69,Z 237.17,A -85,B 0,C 180,E1 23016.623,E2 23016.623} C_VEL
LIN {X 0,Y 496.696,Z 237.177,A -85,B 0,C 180,E1 23013.068,E2 23013.068} C_VEL
LIN {X 0,Y 496.759,Z 237.166,A -85,B 0,C 180,E1 23009.655,E2 23009.655} C_VEL
LIN {X 0,Y 496.697,Z 237.179,A -85,B 0,C 180,E1 23006.237,E2 23006.237} C_VEL
LIN {X 0,Y 496.69,Z 237.182,A -85,B 0,C 180,E1 23002.667,E2 23002.667} C_VEL
LIN {X 0,Y 496.774,Z 237.403,A -85,B 0,C 180,E1 23001.608,E2 23001.608} C_VEL
LIN {X 0,Y 497.191,Z 238.966,A -85,B 0,C 180,E1 23001.36,E2 23001.36} C_VEL
LIN {X 0,Y 499.629,Z 243.284,A -85,B 0,C 180,E1 23000.774,E2 23000.774} C_VEL
LIN {X 0,Y 505.092,Z 253.173,A -85,B 0,C 180,E1 22999.511,E2 22999.511} C_VEL
LIN {X 0,Y 513.043,Z 268.04,A -85,B 0,C 180,E1 22997.778,E2 22997.778} C_VEL
LIN {X 0,Y 519.425,Z 280.001,A -85,B 0,C 180,E1 22996.477,E2 22996.477} C_VEL
LIN {X 0,Y 518.167,Z 316.762,A -85,B 0,C 180,E1 22994.63,E2 22994.63} C_VEL
LIN {X 0,Y 520.099,Z 332.957,A -85,B 0,C 180,E1 22994.214,E2 22994.214} C_VEL
LIN {X 0,Y 518.072,Z 541.876,A -85,B 0,C 180,E1 22991.001,E2 22991.001} C_VEL
LIN {X 0,Y 516.716,Z 655.187,A -85,B 0,C 180,E1 22989.256,E2 22989.256} C_VEL
LIN {X 0,Y 515.905,Z 677.074,A -85,B 0,C 180,E1 22988.799,E2 22988.799} C_VEL
LIN {X 0,Y 514.72,Z 700.419,A -85,B 0,C 180,E1 22988.097,E2 22988.097} C_VEL
LIN {X 0,Y 513.475,Z 719.927,A -85,B 0,C 180,E1 22987.34,E2 22987.34} C_VEL
LIN {X 0,Y 511.702,Z 742.947,A -85,B 0,C 180,E1 22986.225,E2 22986.225} C_VEL
LIN {X 0,Y 509.943,Z 763.957,A -85,B 0,C 180,E1 22984.987,E2 22984.987} C_VEL
LIN {X 0,Y 508.067,Z 783.975,A -85,B 0,C 180,E1 22983.571,E2 22983.571} C_VEL
LIN {X 0,Y 506.161,Z 803.606,A -85,B 0,C 180,E1 22981.963,E2 22981.963} C_VEL
LIN {X 0,Y 504.299,Z 822.141,A -85,B 0,C 180,E1 22980.181,E2 22980.181} C_VEL
LIN {X 0,Y 502.397,Z 841.097,A -85,B 0,C 180,E1 22978.077,E2 22978.077} C_VEL
LIN {X 0,Y 500.864,Z 857.438,A -85,B 0,C 180,E1 22975.986,E2 22975.986} C_VEL
LIN {X 0,Y 499.48,Z 872.669,A -85,B 0,C 180,E1 22973.724,E2 22973.724} C_VEL
LIN {X 0,Y 498.317,Z 886.906,A -85,B 0,C 180,E1 22971.294,E2 22971.294} C_VEL
LIN {X 0,Y 497.484,Z 898.451,A -85,B 0,C 180,E1 22969,E2 22969} C_VEL
LIN {X 0,Y 496.82,Z 909.777,A -85,B 0,C 180,E1 22966.363,E2 22966.363} C_VEL
LIN {X 0,Y 496.404,Z 918.778,A -85,B 0,C 180,E1 22963.867,E2 22963.867} C_VEL
LIN {X 0,Y 496.118,Z 926.354,A -85,B 0,C 180,E1 22961.272,E2 22961.272} C_VEL
LIN {X 0,Y 495.984,Z 932.102,A -85,B 0,C 180,E1 22958.812,E2 22958.812} C_VEL
LIN {X 0,Y 495.933,Z 936.482,A -85,B 0,C 180,E1 22956.249,E2 22956.249} C_VEL
LIN {X 0,Y 495.912,Z 939.183,A -85,B 0,C 180,E1 22953.93,E2 22953.93} C_VEL
LIN {X 0,Y 495.91,Z 940.76,A -85,B 0,C 180,E1 22951.27,E2 22951.27} C_VEL
LIN {X 0,Y 495.913,Z 940.804,A -85,B 0,C 180,E1 22948.959,E2 22948.959} C_VEL
LIN {X 0,Y 495.911,Z 939.406,A -85,B 0,C 180,E1 22946.3,E2 22946.3} C_VEL
LIN {X 0,Y 495.928,Z 936.638,A -85,B 0,C 180,E1 22943.865,E2 22943.865} C_VEL
LIN {X 0,Y 495.982,Z 932.351,A -85,B 0,C 180,E1 22941.303,E2 22941.303} C_VEL
LIN {X 0,Y 496.108,Z 926.65,A -85,B 0,C 180,E1 22938.843,E2 22938.843} C_VEL
LIN {X 0,Y 496.39,Z 919.173,A -85,B 0,C 180,E1 22936.249,E2 22936.249} C_VEL
LIN {X 0,Y 496.798,Z 910.188,A -85,B 0,C 180,E1 22933.742,E2 22933.742} C_VEL
LIN {X 0,Y 497.451,Z 899.015,A -85,B 0,C 180,E1 22931.118,E2 22931.118} C_VEL
LIN {X 0,Y 498.273,Z 887.537,A -85,B 0,C 180,E1 22928.825,E2 22928.825} C_VEL
LIN {X 0,Y 499.418,Z 873.423,A -85,B 0,C 180,E1 22926.395,E2 22926.395} C_VEL
LIN {X 0,Y 500.733,Z 858.738,A -85,B 0,C 180,E1 22924.195,E2 22924.195} C_VEL
LIN {X 0,Y 502.257,Z 842.595,A -85,B 0,C 180,E1 22922.106,E2 22922.106} C_VEL
LIN {X 0,Y 504.037,Z 824.873,A -85,B 0,C 180,E1 22920.098,E2 22920.098} C_VEL
LIN {X 0,Y 505.819,Z 806.911,A -85,B 0,C 180,E1 22918.343,E2 22918.343} C_VEL
LIN {X 0,Y 507.859,Z 786.096,A -85,B 0,C 180,E1 22916.591,E2 22916.591} C_VEL
LIN {X 0,Y 509.706,Z 766.618,A -85,B 0,C 180,E1 22915.191,E2 22915.191} C_VEL
LIN {X 0,Y 511.521,Z 745.051,A -85,B 0,C 180,E1 22913.889,E2 22913.889} C_VEL
LIN {X 0,Y 513.283,Z 722.967,A -85,B 0,C 180,E1 22912.789,E2 22912.789} C_VEL
LIN {X 0,Y 514.638,Z 701.804,A -85,B 0,C 180,E1 22911.952,E2 22911.952} C_VEL
LIN {X 0,Y 515.817,Z 679.763,A -85,B 0,C 180,E1 22911.267,E2 22911.267} C_VEL
LIN {X 0,Y 516.658,Z 657.06,A -85,B 0,C 180,E1 22910.778,E2 22910.778} C_VEL
LIN {X 0,Y 518.39,Z 524.095,A -85,B 0,C 180,E1 22908.706,E2 22908.706} C_VEL
LIN {X 0,Y 520.552,Z 331.003,A -85,B 0,C 180,E1 22905.673,E2 22905.673} C_VEL
LIN {X 0,Y 518.575,Z 314.312,A -85,B 0,C 180,E1 22905.197,E2 22905.197} C_VEL
LIN {X 0,Y 520.015,Z 280.231,A -85,B 0,C 180,E1 22903.423,E2 22903.423} C_VEL
LIN {X 0,Y 508.68,Z 259.299,A -85,B 0,C 180,E1 22901.034,E2 22901.034} C_VEL
LIN {X 0,Y 501.317,Z 246.148,A -85,B 0,C 180,E1 22899.364,E2 22899.364} C_VEL
LIN {X 0,Y 498.626,Z 241.4,A -85,B 0,C 180,E1 22898.729,E2 22898.729} C_VEL
LIN {X 0,Y 496.804,Z 237.693,A -85,B 0,C 180,E1 22898.222,E2 22898.222} C_VEL
LIN {X 0,Y 496.697,Z 237.171,A -85,B 0,C 180,E1 22897.877,E2 22897.877} C_VEL
LIN {X 0,Y 496.751,Z 237.162,A -85,B 0,C 180,E1 22894.444,E2 22894.444} C_VEL
LIN {X 0,Y 496.711,Z 237.171,A -85,B 0,C 180,E1 22891.019,E2 22891.019} C_VEL
LIN {X 0,Y 496.707,Z 237.175,A -85,B 0,C 180,E1 22887.58,E2 22887.58} C_VEL
LIN {X 0,Y 496.758,Z 237.172,A -85,B 0,C 180,E1 22884.117,E2 22884.117} C_VEL
LIN {X 0,Y 496.726,Z 237.171,A -85,B 0,C 180,E1 22880.749,E2 22880.749} C_VEL
LIN {X 0,Y 496.714,Z 237.171,A -85,B 0,C 180,E1 22877.212,E2 22877.212} C_VEL
LIN {X 0,Y 496.751,Z 237.165,A -85,B 0,C 180,E1 22873.74,E2 22873.74} C_VEL
LIN {X 0,Y 496.748,Z 237.16,A -85,B 0,C 180,E1 22870.32,E2 22870.32} C_VEL
LIN {X 0,Y 496.718,Z 237.169,A -85,B 0,C 180,E1 22866.937,E2 22866.937} C_VEL
LIN {X 0,Y 496.754,Z 237.168,A -85,B 0,C 180,E1 22863.462,E2 22863.462} C_VEL
LIN {X 0,Y 496.773,Z 237.161,A -85,B 0,C 180,E1 22859.885,E2 22859.885} C_VEL
LIN {X 0,Y 496.732,Z 237.16,A -85,B 0,C 180,E1 22856.423,E2 22856.423} C_VEL
LIN {X 0,Y 496.736,Z 237.167,A -85,B 0,C 180,E1 22852.831,E2 22852.831} C_VEL
LIN {X 0,Y 496.769,Z 237.167,A -85,B 0,C 180,E1 22849.329,E2 22849.329} C_VEL
LIN {X 0,Y 496.766,Z 237.155,A -85,B 0,C 180,E1 22845.786,E2 22845.786} C_VEL
LIN {X 0,Y 496.74,Z 237.169,A -85,B 0,C 180,E1 22842.306,E2 22842.306} C_VEL
LIN {X 0,Y 496.759,Z 237.165,A -85,B 0,C 180,E1 22838.736,E2 22838.736} C_VEL
LIN {X 0,Y 496.765,Z 237.157,A -85,B 0,C 180,E1 22835.197,E2 22835.197} C_VEL
LIN {X 0,Y 496.768,Z 237.161,A -85,B 0,C 180,E1 22831.591,E2 22831.591} C_VEL
LIN {X 0,Y 496.752,Z 237.168,A -85,B 0,C 180,E1 22828.038,E2 22828.038} C_VEL
LIN {X 0,Y 496.765,Z 237.159,A -85,B 0,C 180,E1 22824.574,E2 22824.574} C_VEL
LIN {X 0,Y 496.76,Z 237.155,A -85,B 0,C 180,E1 22820.981,E2 22820.981} C_VEL
LIN {X 0,Y 496.763,Z 237.169,A -85,B 0,C 180,E1 22817.447,E2 22817.447} C_VEL
LIN {X 0,Y 496.76,Z 237.166,A -85,B 0,C 180,E1 22813.821,E2 22813.821} C_VEL
LIN {X 0,Y 496.765,Z 237.163,A -85,B 0,C 180,E1 22810.248,E2 22810.248} C_VEL
LIN {X 0,Y 496.754,Z 237.162,A -85,B 0,C 180,E1 22806.713,E2 22806.713} C_VEL
LIN {X 0,Y 496.76,Z 237.164,A -85,B 0,C 180,E1 22806.204,E2 22806.204} C_VEL
LIN {X 0,Y 495.789,Z 237.292,A -85,B 0,C 180,E1 22805.315,E2 22805.315} C_VEL
LIN {X 0,Y 489.332,Z 238.093,A -85,B 0,C 180,E1 22802.818,E2 22802.818} C_VEL
LIN {X 0,Y 488.818,Z 238.156,A -85,B 0,C 180,E1 22802.166,E2 22802.166} C_VEL
LIN {X 0,Y 488.814,Z 238.158,A -85,B 0,C 180,E1 22798.598,E2 22798.598} C_VEL
LIN {X 0,Y 488.831,Z 238.157,A -85,B 0,C 180,E1 22795.028,E2 22795.028} C_VEL
LIN {X 0,Y 488.825,Z 238.11,A -85,B 0,C 180,E1 22791.352,E2 22791.352} C_VEL
LIN {X 0,Y 488.805,Z 238.129,A -85,B 0,C 180,E1 22787.869,E2 22787.869} C_VEL
LIN {X 0,Y 488.849,Z 238.387,A -85,B 0,C 180,E1 22786.549,E2 22786.549} C_VEL
LIN {X 0,Y 490.106,Z 241.609,A -85,B 0,C 180,E1 22786.082,E2 22786.082} C_VEL
LIN {X 0,Y 491.374,Z 243.855,A -85,B 0,C 180,E1 22785.75,E2 22785.75} C_VEL
LIN {X 0,Y 499.699,Z 260.61,A -85,B 0,C 180,E1 22783.485,E2 22783.485} C_VEL
LIN {X 0,Y 507.41,Z 277.303,A -85,B 0,C 180,E1 22781.423,E2 22781.423} C_VEL
LIN {X 0,Y 503.938,Z 331.247,A -85,B 0,C 180,E1 22777.812,E2 22777.812} C_VEL
LIN {X 0,Y 500.883,Z 384.85,A -85,B 0,C 180,E1 22774.294,E2 22774.294} C_VEL
LIN {X 0,Y 499.661,Z 411.162,A -85,B 0,C 180,E1 22772.621,E2 22772.621} C_VEL
LIN {X 0,Y 502.302,Z 433.481,A -85,B 0,C 180,E1 22772.017,E2 22772.017} C_VEL
LIN {X 0,Y 498.794,Z 630.377,A -85,B 0,C 180,E1 22768.845,E2 22768.845} C_VEL
LIN {X 0,Y 498.073,Z 649.826,A -85,B 0,C 180,E1 22768.315,E2 22768.315} C_VEL
LIN {X 0,Y 497.24,Z 667.288,A -85,B 0,C 180,E1 22767.639,E2 22767.639} C_VEL
LIN {X 0,Y 496.172,Z 685.455,A -85,B 0,C 180,E1 22766.709,E2 22766.709} C_VEL
LIN {X 0,Y 494.997,Z 702.54,A -85,B 0,C 180,E1 22765.599,E2 22765.599} C_VEL
LIN {X 0,Y 493.782,Z 718.647,A -85,B 0,C 180,E1 22764.307,E2 22764.307} C_VEL
LIN {X 0,Y 492.586,Z 733.772,A -85,B 0,C 180,E1 22762.83,E2 22762.83} C_VEL
LIN {X 0,Y 491.483,Z 747.41,A -85,B 0,C 180,E1 22761.225,E2 22761.225} C_VEL
LIN {X 0,Y 490.555,Z 759.299,A -85,B 0,C 180,E1 22759.55,E2 22759.55} C_VEL
LIN {X 0,Y 489.723,Z 770.604,A -85,B 0,C 180,E1 22757.622,E2 22757.622} C_VEL
LIN {X 0,Y 489.1,Z 779.938,A -85,B 0,C 180,E1 22755.68,E2 22755.68} C_VEL
LIN {X 0,Y 488.658,Z 787.954,A -85,B 0,C 180,E1 22753.6,E2 22753.6} C_VEL
LIN {X 0,Y 488.362,Z 794.42,A -85,B 0,C 180,E1 22751.427,E2 22751.427} C_VEL
LIN {X 0,Y 488.199,Z 799.132,A -85,B 0,C 180,E1 22749.25,E2 22749.25} C_VEL
LIN {X 0,Y 488.135,Z 802.169,A -85,B 0,C 180,E1 22747.098,E2 22747.098} C_VEL
LIN {X 0,Y 488.112,Z 803.678,A -85,B 0,C 180,E1 22744.875,E2 22744.875} C_VEL
LIN {X 0,Y 488.116,Z 803.599,A -85,B 0,C 180,E1 22742.689,E2 22742.689} C_VEL
LIN {X 0,Y 488.158,Z 801.849,A -85,B 0,C 180,E1 22740.423,E2 22740.423} C_VEL
LIN {X 0,Y 488.261,Z 798.456,A -85,B 0,C 180,E1 22738.192,E2 22738.192} C_VEL
LIN {X 0,Y 488.473,Z 793.403,A -85,B 0,C 180,E1 22735.994,E2 22735.994} C_VEL
LIN {X 0,Y 488.8,Z 786.894,A -85,B 0,C 180,E1 22733.898,E2 22733.898} C_VEL
LIN {X 0,Y 489.295,Z 778.894,A -85,B 0,C 180,E1 22731.88,E2 22731.88} C_VEL
LIN {X 0,Y 490.004,Z 769.274,A -85,B 0,C 180,E1 22729.923,E2 22729.923} C_VEL
LIN {X 0,Y 490.892,Z 757.879,A -85,B 0,C 180,E1 22728.024,E2 22728.024} C_VEL
LIN {X 0,Y 491.961,Z 745.301,A -85,B 0,C 180,E1 22726.292,E2 22726.292} C_VEL
LIN {X 0,Y 493.133,Z 731.518,A -85,B 0,C 180,E1 22724.713,E2 22724.713} C_VEL
LIN {X 0,Y 494.384,Z 716.414,A -85,B 0,C 180,E1 22723.277,E2 22723.277} C_VEL
LIN {X 0,Y 495.616,Z 700.745,A -85,B 0,C 180,E1 22722.049,E2 22722.049} C_VEL
LIN {X 0,Y 496.844,Z 683.729,A -85,B 0,C 180,E1 22720.968,E2 22720.968} C_VEL
LIN {X 0,Y 497.923,Z 666.272,A -85,B 0,C 180,E1 22720.089,E2 22720.089} C_VEL
LIN {X 0,Y 498.846,Z 647.761,A -85,B 0,C 180,E1 22719.386,E2 22719.386} C_VEL
LIN {X 0,Y 499.584,Z 628.694,A -85,B 0,C 180,E1 22718.886,E2 22718.886} C_VEL
LIN {X 0,Y 503.733,Z 431.903,A -85,B 0,C 180,E1 22715.622,E2 22715.622} C_VEL
LIN {X 0,Y 500.719,Z 407.188,A -85,B 0,C 180,E1 22714.848,E2 22714.848} C_VEL
LIN {X 0,Y 504.286,Z 348.286,A -85,B 0,C 180,E1 22710.964,E2 22710.964} C_VEL
LIN {X 0,Y 508.036,Z 294.848,A -85,B 0,C 180,E1 22707.364,E2 22707.364} C_VEL
LIN {X 0,Y 509.05,Z 279.38,A -85,B 0,C 180,E1 22706.29,E2 22706.29} C_VEL
LIN {X 0,Y 500.253,Z 260.651,A -85,B 0,C 180,E1 22703.811,E2 22703.811} C_VEL
LIN {X 0,Y 493.071,Z 246.942,A -85,B 0,C 180,E1 22701.766,E2 22701.766} C_VEL
LIN {X 0,Y 490.557,Z 242.21,A -85,B 0,C 180,E1 22701.021,E2 22701.021} C_VEL
LIN {X 0,Y 488.838,Z 238.641,A -85,B 0,C 180,E1 22700.441,E2 22700.441} C_VEL
LIN {X 0,Y 488.749,Z 238.155,A -85,B 0,C 180,E1 22700.101,E2 22700.101} C_VEL
LIN {X 0,Y 488.786,Z 238.159,A -85,B 0,C 180,E1 22696.641,E2 22696.641} C_VEL
LIN {X 0,Y 488.769,Z 238.167,A -85,B 0,C 180,E1 22693.365,E2 22693.365} C_VEL
LIN {X 0,Y 488.749,Z 238.162,A -85,B 0,C 180,E1 22689.894,E2 22689.894} C_VEL
LIN {X 0,Y 488.797,Z 238.164,A -85,B 0,C 180,E1 22686.459,E2 22686.459} C_VEL
LIN {X 0,Y 488.767,Z 238.164,A -85,B 0,C 180,E1 22683.048,E2 22683.048} C_VEL
LIN {X 0,Y 488.748,Z 238.158,A -85,B 0,C 180,E1 22679.648,E2 22679.648} C_VEL
LIN {X 0,Y 488.8,Z 238.157,A -85,B 0,C 180,E1 22676.247,E2 22676.247} C_VEL
LIN {X 0,Y 488.765,Z 238.162,A -85,B 0,C 180,E1 22672.804,E2 22672.804} C_VEL
LIN {X 0,Y 488.746,Z 238.166,A -85,B 0,C 180,E1 22669.271,E2 22669.271} C_VEL
LIN {X 0,Y 488.782,Z 238.158,A -85,B 0,C 180,E1 22665.79,E2 22665.79} C_VEL
